LIN {X 0,Y 523.586,Z 1035.497,A -85,B 0,C 180,E1 24820.361,E2 24820.361} C_VEL
LIN {X 0,Y 523.955,Z 1017.547,A -85,B 0,C 180,E1 24819.86,E2 24819.86} C_VEL
LIN {X 0,Y 524.216,Z 988.491,A -85,B 0,C 180,E1 24819.409,E2 24819.409} C_VEL
LIN {X 0,Y 525.099,Z 854.259,A -85,B 0,C 180,E1 24817.476,E2 24817.476} C_VEL
LIN {X 0,Y 524.353,Z 848.699,A -85,B 0,C 180,E1 24817.345,E2 24817.345} C_VEL
LIN {X 0,Y 527.314,Z 813.157,A -85,B 0,C 180,E1 24813.997,E2 24813.997} C_VEL
LIN {X 0,Y 530.511,Z 784.43,A -85,B 0,C 180,E1 24811.152,E2 24811.152} C_VEL
LIN {X 0,Y 534.459,Z 760.277,A -85,B 0,C 180,E1 24808.6,E2 24808.6} C_VEL
LIN {X 0,Y 539.863,Z 738.188,A -85,B 0,C 180,E1 24806.071,E2 24806.071} C_VEL
LIN {X 0,Y 545.29,Z 723.44,A -85,B 0,C 180,E1 24804.202,E2 24804.202} C_VEL
LIN {X 0,Y 548.271,Z 717.496,A -85,B 0,C 180,E1 24803.361,E2 24803.361} C_VEL
LIN {X 0,Y 540.635,Z 729.193,A -85,B 0,C 180,E1 24802.158,E2 24802.158} C_VEL
LIN {X 0,Y 535.477,Z 740.888,A -85,B 0,C 180,E1 24801.051,E2 24801.051} C_VEL
LIN {X 0,Y 532.179,Z 753.467,A -85,B 0,C 180,E1 24799.962,E2 24799.962} C_VEL
LIN {X 0,Y 530.634,Z 767.779,A -85,B 0,C 180,E1 24798.804,E2 24798.804} C_VEL
LIN {X 0,Y 531.093,Z 781.511,A -85,B 0,C 180,E1 24797.721,E2 24797.721} C_VEL
LIN {X 0,Y 533.486,Z 794.423,A -85,B 0,C 180,E1 24796.689,E2 24796.689} C_VEL
LIN {X 0,Y 537.671,Z 806.101,A -85,B 0,C 180,E1 24795.721,E2 24795.721} C_VEL
LIN {X 0,Y 543.177,Z 815.91,A -85,B 0,C 180,E1 24794.872,E2 24794.872} C_VEL
LIN {X 0,Y 550.682,Z 825.132,A -85,B 0,C 180,E1 24794.028,E2 24794.028} C_VEL
LIN {X 0,Y 559.874,Z 833.081,A -85,B 0,C 180,E1 24793.229,E2 24793.229} C_VEL
LIN {X 0,Y 568.972,Z 838.703,A -85,B 0,C 180,E1 24792.582,E2 24792.582} C_VEL
LIN {X 0,Y 573.371,Z 840.473,A -85,B 0,C 180,E1 24792.173,E2 24792.173} C_VEL
LIN {X 0,Y 577.044,Z 841.244,A -85,B 0,C 180,E1 24791.686,E2 24791.686} C_VEL
LIN {X 0,Y 579.923,Z 840.965,A -85,B 0,C 180,E1 24791.111,E2 24791.111} C_VEL
LIN {X 0,Y 581.493,Z 839.74,A -85,B 0,C 180,E1 24790.536,E2 24790.536} C_VEL
LIN {X 0,Y 581.774,Z 837.458,A -85,B 0,C 180,E1 24789.918,E2 24789.918} C_VEL
LIN {X 0,Y 580.503,Z 834.257,A -85,B 0,C 180,E1 24789.335,E2 24789.335} C_VEL
LIN {X 0,Y 577.813,Z 830.456,A -85,B 0,C 180,E1 24788.85,E2 24788.85} C_VEL
LIN {X 0,Y 571.058,Z 821.059,A -85,B 0,C 180,E1 24788,E2 24788} C_VEL
LIN {X 0,Y 565.628,Z 811.116,A -85,B 0,C 180,E1 24787.29,E2 24787.29} C_VEL
LIN {X 0,Y 561.482,Z 850.258,A -85,B 0,C 180,E1 24786.731,E2 24786.731} C_VEL
LIN {X 0,Y 558.358,Z 872.045,A -85,B 0,C 180,E1 24786.299,E2 24786.299} C_VEL
LIN {X 0,Y 556.202,Z 881.325,A -85,B 0,C 180,E1 24785.996,E2 24785.996} C_VEL
LIN {X 0,Y 555.687,Z 885.783,A -85,B 0,C 180,E1 24785.923,E2 24785.923} C_VEL
LIN {X 0,Y 552.428,Z 921.98,A -85,B 0,C 180,E1 24785.512,E2 24785.512} C_VEL
LIN {X 0,Y 548.555,Z 944.063,A -85,B 0,C 180,E1 24785.284,E2 24785.284} C_VEL
LIN {X 0,Y 544.213,Z 961.518,A -85,B 0,C 180,E1 24784.984,E2 24784.984} C_VEL
LIN {X 0,Y 541.11,Z 972.645,A -85,B 0,C 180,E1 24784.625,E2 24784.625} C_VEL
LIN {X 0,Y 540.107,Z 976.205,A -85,B 0,C 180,E1 24784.487,E2 24784.487} C_VEL
LIN {X 0,Y 536.14,Z 989.922,A -85,B 0,C 180,E1 24784.214,E2 24784.214} C_VEL
LIN {X 0,Y 533.243,Z 1000.027,A -85,B 0,C 180,E1 24783.841,E2 24783.841} C_VEL
LIN {X 0,Y 532.563,Z 1003.315,A -85,B 0,C 180,E1 24783.7,E2 24783.7} C_VEL
LIN {X 0,Y 531.76,Z 1066.201,A -85,B 0,C 180,E1 24782.724,E2 24782.724} C_VEL
LIN {X 0,Y 531.071,Z 1087.988,A -85,B 0,C 180,E1 24782.192,E2 24782.192} C_VEL
LIN {X 0,Y 530.194,Z 1110.298,A -85,B 0,C 180,E1 24781.429,E2 24781.429} C_VEL
LIN {X 0,Y 529.157,Z 1131.269,A -85,B 0,C 180,E1 24780.501,E2 24780.501} C_VEL
LIN {X 0,Y 528.011,Z 1151.791,A -85,B 0,C 180,E1 24779.371,E2 24779.371} C_VEL
LIN {X 0,Y 526.773,Z 1171.709,A -85,B 0,C 180,E1 24778.042,E2 24778.042} C_VEL
LIN {X 0,Y 525.528,Z 1191.133,A -85,B 0,C 180,E1 24776.498,E2 24776.498} C_VEL
LIN {X 0,Y 524.371,Z 1208.653,A -85,B 0,C 180,E1 24774.857,E2 24774.857} C_VEL
LIN {X 0,Y 523.398,Z 1223.625,A -85,B 0,C 180,E1 24773.24,E2 24773.24} C_VEL
LIN {X 0,Y 522.415,Z 1239.904,A -85,B 0,C 180,E1 24771.207,E2 24771.207} C_VEL
LIN {X 0,Y 521.625,Z 1254.014,A -85,B 0,C 180,E1 24769.134,E2 24769.134} C_VEL
LIN {X 0,Y 521.016,Z 1266.743,A -85,B 0,C 180,E1 24766.96,E2 24766.96} C_VEL
LIN {X 0,Y 520.548,Z 1277.844,A -85,B 0,C 180,E1 24764.688,E2 24764.688} C_VEL
LIN {X 0,Y 520.249,Z 1287.1,A -85,B 0,C 180,E1 24762.431,E2 24762.431} C_VEL
LIN {X 0,Y 520.058,Z 1295.215,A -85,B 0,C 180,E1 24759.965,E2 24759.965} C_VEL
LIN {X 0,Y 519.971,Z 1300.895,A -85,B 0,C 180,E1 24757.736,E2 24757.736} C_VEL
LIN {X 0,Y 519.921,Z 1305.493,A -85,B 0,C 180,E1 24755.297,E2 24755.297} C_VEL
LIN {X 0,Y 519.902,Z 1308.295,A -85,B 0,C 180,E1 24752.867,E2 24752.867} C_VEL
LIN {X 0,Y 519.896,Z 1309.373,A -85,B 0,C 180,E1 24750.662,E2 24750.662} C_VEL
LIN {X 0,Y 519.896,Z 1309.038,A -85,B 0,C 180,E1 24748.237,E2 24748.237} C_VEL
LIN {X 0,Y 519.905,Z 1307.108,A -85,B 0,C 180,E1 24745.92,E2 24745.92} C_VEL
LIN {X 0,Y 519.931,Z 1303.619,A -85,B 0,C 180,E1 24743.597,E2 24743.597} C_VEL
LIN {X 0,Y 519.999,Z 1298.291,A -85,B 0,C 180,E1 24741.152,E2 24741.152} C_VEL
LIN {X 0,Y 520.135,Z 1291.394,A -85,B 0,C 180,E1 24738.805,E2 24738.805} C_VEL
LIN {X 0,Y 520.382,Z 1282.793,A -85,B 0,C 180,E1 24736.463,E2 24736.463} C_VEL
LIN {X 0,Y 520.771,Z 1271.951,A -85,B 0,C 180,E1 24734.065,E2 24734.065} C_VEL
LIN {X 0,Y 521.239,Z 1261.598,A -85,B 0,C 180,E1 24732.127,E2 24732.127} C_VEL
LIN {X 0,Y 521.949,Z 1248.058,A -85,B 0,C 180,E1 24729.947,E2 24729.947} C_VEL
LIN {X 0,Y 522.774,Z 1233.701,A -85,B 0,C 180,E1 24727.984,E2 24727.984} C_VEL
LIN {X 0,Y 523.673,Z 1219.46,A -85,B 0,C 180,E1 24726.288,E2 24726.288} C_VEL
LIN {X 0,Y 524.839,Z 1201.727,A -85,B 0,C 180,E1 24724.459,E2 24724.459} C_VEL
LIN {X 0,Y 526.047,Z 1182.855,A -85,B 0,C 180,E1 24722.814,E2 24722.814} C_VEL
LIN {X 0,Y 527.349,Z 1162.825,A -85,B 0,C 180,E1 24721.336,E2 24721.336} C_VEL
LIN {X 0,Y 528.528,Z 1142.749,A -85,B 0,C 180,E1 24720.101,E2 24720.101} C_VEL
LIN {X 0,Y 529.657,Z 1121.584,A -85,B 0,C 180,E1 24719.043,E2 24719.043} C_VEL
LIN {X 0,Y 530.645,Z 1099.656,A -85,B 0,C 180,E1 24718.181,E2 24718.181} C_VEL
LIN {X 0,Y 531.428,Z 1077.651,A -85,B 0,C 180,E1 24717.53,E2 24717.53} C_VEL
LIN {X 0,Y 531.973,Z 1055.21,A -85,B 0,C 180,E1 24717.082,E2 24717.082} C_VEL
LIN {X 0,Y 532.624,Z 1002.328,A -85,B 0,C 180,E1 24716.277,E2 24716.277} C_VEL
LIN {X 0,Y 535.397,Z 992.455,A -85,B 0,C 180,E1 24715.863,E2 24715.863} C_VEL
LIN {X 0,Y 539.286,Z 979.138,A -85,B 0,C 180,E1 24715.554,E2 24715.554} C_VEL
LIN {X 0,Y 540.609,Z 974.405,A -85,B 0,C 180,E1 24715.46,E2 24715.46} C_VEL
LIN {X 0,Y 543.293,Z 964.872,A -85,B 0,C 180,E1 24715.102,E2 24715.102} C_VEL
LIN {X 0,Y 547.461,Z 948.839,A -85,B 0,C 180,E1 24714.78,E2 24714.78} C_VEL
LIN {X 0,Y 551.573,Z 927.951,A -85,B 0,C 180,E1 24714.547,E2 24714.547} C_VEL
LIN {X 0,Y 554.193,Z 904.712,A -85,B 0,C 180,E1 24714.291,E2 24714.291} C_VEL
LIN {X 0,Y 556.16,Z 881.458,A -85,B 0,C 180,E1 24714.01,E2 24714.01} C_VEL
LIN {X 0,Y 558.316,Z 872.279,A -85,B 0,C 180,E1 24713.707,E2 24713.707} C_VEL
LIN {X 0,Y 561.42,Z 850.756,A -85,B 0,C 180,E1 24713.277,E2 24713.277} C_VEL
LIN {X 0,Y 565.558,Z 811.884,A -85,B 0,C 180,E1 24712.719,E2 24712.719} C_VEL
LIN {X 0,Y 565.709,Z 810.985,A -85,B 0,C 180,E1 24712.699,E2 24712.699} C_VEL
LIN {X 0,Y 571.284,Z 821.421,A -85,B 0,C 180,E1 24711.971,E2 24711.971} C_VEL
LIN {X 0,Y 577.959,Z 830.632,A -85,B 0,C 180,E1 24711.131,E2 24711.131} C_VEL
LIN {X 0,Y 580.567,Z 834.367,A -85,B 0,C 180,E1 24710.648,E2 24710.648} C_VEL
LIN {X 0,Y 581.789,Z 837.556,A -85,B 0,C 180,E1 24710.061,E2 24710.061} C_VEL
LIN {X 0,Y 581.489,Z 839.748,A -85,B 0,C 180,E1 24709.462,E2 24709.462} C_VEL
LIN {X 0,Y 579.921,Z 840.971,A -85,B 0,C 180,E1 24708.889,E2 24708.889} C_VEL
LIN {X 0,Y 577.042,Z 841.249,A -85,B 0,C 180,E1 24708.314,E2 24708.314} C_VEL
LIN {X 0,Y 573.37,Z 840.478,A -85,B 0,C 180,E1 24707.827,E2 24707.827} C_VEL
LIN {X 0,Y 564.453,Z 836.474,A -85,B 0,C 180,E1 24706.87,E2 24706.87} C_VEL
LIN {X 0,Y 556.319,Z 830.523,A -85,B 0,C 180,E1 24705.816,E2 24705.816} C_VEL
LIN {X 0,Y 549.697,Z 823.015,A -85,B 0,C 180,E1 24704.742,E2 24704.742} C_VEL
LIN {X 0,Y 544.58,Z 813.966,A -85,B 0,C 180,E1 24703.657,E2 24703.657} C_VEL
LIN {X 0,Y 540.972,Z 803.368,A -85,B 0,C 180,E1 24702.568,E2 24702.568} C_VEL
LIN {X 0,Y 538.865,Z 790.955,A -85,B 0,C 180,E1 24701.444,E2 24701.444} C_VEL
LIN {X 0,Y 538.28,Z 775.777,A -85,B 0,C 180,E1 24700.233,E2 24700.233} C_VEL
LIN {X 0,Y 541.066,Z 725.504,A -85,B 0,C 180,E1 24696.581,E2 24696.581} C_VEL
LIN {X 0,Y 541.898,Z 709.421,A -85,B 0,C 180,E1 24695.361,E2 24695.361} C_VEL
LIN {X 0,Y 533.055,Z 693.053,A -85,B 0,C 180,E1 24692.825,E2 24692.825} C_VEL
LIN {X 0,Y 527.803,Z 683.663,A -85,B 0,C 180,E1 24691.269,E2 24691.269} C_VEL
LIN {X 0,Y 525.459,Z 679.281,A -85,B 0,C 180,E1 24690.534,E2 24690.534} C_VEL
LIN {X 0,Y 523.439,Z 675.653,A -85,B 0,C 180,E1 24689.904,E2 24689.904} C_VEL
LIN {X 0,Y 522.358,Z 673.996,A -85,B 0,C 180,E1 24689.593,E2 24689.593} C_VEL
LIN {X 0,Y 520.765,Z 670.882,A -85,B 0,C 180,E1 24689.062,E2 24689.062} C_VEL
LIN {X 0,Y 520.584,Z 669.89,A -85,B 0,C 180,E1 24688.904,E2 24688.904} C_VEL
LIN {X 0,Y 520.583,Z 669.888,A -85,B 0,C 180,E1 24685.36,E2 24685.36} C_VEL
LIN {X 0,Y 520.582,Z 669.887,A -85,B 0,C 180,E1 24681.876,E2 24681.876} C_VEL
LIN {X 0,Y 520.574,Z 669.89,A -85,B 0,C 180,E1 24678.413,E2 24678.413} C_VEL
LIN {X 0,Y 520.583,Z 669.892,A -85,B 0,C 180,E1 24674.967,E2 24674.967} C_VEL
LIN {X 0,Y 520.588,Z 669.889,A -85,B 0,C 180,E1 24671.41,E2 24671.41} C_VEL
LIN {X 0,Y 520.576,Z 669.889,A -85,B 0,C 180,E1 24667.837,E2 24667.837} C_VEL
LIN {X 0,Y 520.586,Z 669.889,A -85,B 0,C 180,E1 24664.406,E2 24664.406} C_VEL
LIN {X 0,Y 520.586,Z 669.888,A -85,B 0,C 180,E1 24660.88,E2 24660.88} C_VEL
LIN {X 0,Y 520.582,Z 669.889,A -85,B 0,C 180,E1 24657.358,E2 24657.358} C_VEL
LIN {X 0,Y 520.587,Z 669.889,A -85,B 0,C 180,E1 24653.825,E2 24653.825} C_VEL
LIN {X 0,Y 520.587,Z 669.892,A -85,B 0,C 180,E1 24650.269,E2 24650.269} C_VEL
LIN {X 0,Y 520.577,Z 669.888,A -85,B 0,C 180,E1 24646.787,E2 24646.787} C_VEL
LIN {X 0,Y 520.587,Z 669.888,A -85,B 0,C 180,E1 24643.256,E2 24643.256} C_VEL
LIN {X 0,Y 520.582,Z 669.888,A -85,B 0,C 180,E1 24639.657,E2 24639.657} C_VEL
LIN {X 0,Y 520.574,Z 669.889,A -85,B 0,C 180,E1 24636.212,E2 24636.212} C_VEL
LIN {X 0,Y 520.581,Z 669.879,A -85,B 0,C 180,E1 24632.779,E2 24632.779} C_VEL
LIN {X 0,Y 520.589,Z 669.881,A -85,B 0,C 180,E1 24629.277,E2 24629.277} C_VEL
LIN {X 0,Y 520.588,Z 669.876,A -85,B 0,C 180,E1 24625.754,E2 24625.754} C_VEL
LIN {X 0,Y 520.581,Z 669.892,A -85,B 0,C 180,E1 24622.307,E2 24622.307} C_VEL
LIN {X 0,Y 520.571,Z 669.873,A -85,B 0,C 180,E1 24618.842,E2 24618.842} C_VEL
LIN {X 0,Y 520.585,Z 669.882,A -85,B 0,C 180,E1 24617.879,E2 24617.879} C_VEL
LIN {X 0,Y 519.613,Z 670.014,A -85,B 0,C 180,E1 24617.032,E2 24617.032} C_VEL
LIN {X 0,Y 513.091,Z 670.826,A -85,B 0,C 180,E1 24614.588,E2 24614.588} C_VEL
LIN {X 0,Y 512.64,Z 670.882,A -85,B 0,C 180,E1 24614.028,E2 24614.028} C_VEL
LIN {X 0,Y 512.679,Z 671.112,A -85,B 0,C 180,E1 24610.616,E2 24610.616} C_VEL
LIN {X 0,Y 513.821,Z 674.165,A -85,B 0,C 180,E1 24610.288,E2 24610.288} C_VEL
LIN {X 0,Y 522.026,Z 692.981,A -85,B 0,C 180,E1 24608.163,E2 24608.163} C_VEL
LIN {X 0,Y 524.698,Z 700.431,A -85,B 0,C 180,E1 24607.379,E2 24607.379} C_VEL
LIN {X 0,Y 522.968,Z 748.227,A -85,B 0,C 180,E1 24604.002,E2 24604.002} C_VEL
LIN {X 0,Y 522.481,Z 768.097,A -85,B 0,C 180,E1 24602.665,E2 24602.665} C_VEL
LIN {X 0,Y 524.515,Z 781.949,A -85,B 0,C 180,E1 24602.299,E2 24602.299} C_VEL
LIN {X 0,Y 521.936,Z 1016.462,A -85,B 0,C 180,E1 24598.79,E2 24598.79} C_VEL
LIN {X 0,Y 521.472,Z 1038.136,A -85,B 0,C 180,E1 24598.367,E2 24598.367} C_VEL
LIN {X 0,Y 520.771,Z 1058.877,A -85,B 0,C 180,E1 24597.752,E2 24597.752} C_VEL
LIN {X 0,Y 519.953,Z 1077.833,A -85,B 0,C 180,E1 24596.988,E2 24596.988} C_VEL
LIN {X 0,Y 519.007,Z 1096.138,A -85,B 0,C 180,E1 24596.055,E2 24596.055} C_VEL
LIN {X 0,Y 517.914,Z 1115.556,A -85,B 0,C 180,E1 24594.833,E2 24594.833} C_VEL
LIN {X 0,Y 516.831,Z 1133.209,A -85,B 0,C 180,E1 24593.485,E2 24593.485} C_VEL
LIN {X 0,Y 515.776,Z 1149.876,A -85,B 0,C 180,E1 24591.971,E2 24591.971} C_VEL
LIN {X 0,Y 514.806,Z 1165.721,A -85,B 0,C 180,E1 24590.267,E2 24590.267} C_VEL
LIN {X 0,Y 513.937,Z 1180.619,A -85,B 0,C 180,E1 24588.37,E2 24588.37} C_VEL
LIN {X 0,Y 513.248,Z 1193.625,A -85,B 0,C 180,E1 24586.407,E2 24586.407} C_VEL
LIN {X 0,Y 512.723,Z 1205.136,A -85,B 0,C 180,E1 24584.339,E2 24584.339} C_VEL
LIN {X 0,Y 512.365,Z 1214.674,A -85,B 0,C 180,E1 24582.281,E2 24582.281} C_VEL
LIN {X 0,Y 512.118,Z 1223.218,A -85,B 0,C 180,E1 24580.006,E2 24580.006} C_VEL
LIN {X 0,Y 511.993,Z 1229.79,A -85,B 0,C 180,E1 24577.744,E2 24577.744} C_VEL
LIN {X 0,Y 511.93,Z 1234.587,A -85,B 0,C 180,E1 24575.491,E2 24575.491} C_VEL
LIN {X 0,Y 511.913,Z 1237.847,A -85,B 0,C 180,E1 24573.135,E2 24573.135} C_VEL
LIN {X 0,Y 511.91,Z 1239.341,A -85,B 0,C 180,E1 24570.783,E2 24570.783} C_VEL
LIN {X 0,Y 511.9,Z 1239.167,A -85,B 0,C 180,E1 24568.545,E2 24568.545} C_VEL
LIN {X 0,Y 511.911,Z 1237.374,A -85,B 0,C 180,E1 24566.304,E2 24566.304} C_VEL
LIN {X 0,Y 511.938,Z 1233.93,A -85,B 0,C 180,E1 24564.058,E2 24564.058} C_VEL
LIN {X 0,Y 511.996,Z 1228.822,A -85,B 0,C 180,E1 24561.804,E2 24561.804} C_VEL
LIN {X 0,Y 512.143,Z 1221.931,A -85,B 0,C 180,E1 24559.539,E2 24559.539} C_VEL
LIN {X 0,Y 512.406,Z 1213.59,A -85,B 0,C 180,E1 24557.376,E2 24557.376} C_VEL
LIN {X 0,Y 512.812,Z 1203.268,A -85,B 0,C 180,E1 24555.201,E2 24555.201} C_VEL
LIN {X 0,Y 513.373,Z 1191.365,A -85,B 0,C 180,E1 24553.13,E2 24553.13} C_VEL
LIN {X 0,Y 514.102,Z 1177.909,A -85,B 0,C 180,E1 24551.164,E2 24551.164} C_VEL
LIN {X 0,Y 514.959,Z 1163.358,A -85,B 0,C 180,E1 24549.369,E2 24549.369} C_VEL
LIN {X 0,Y 515.916,Z 1147.72,A -85,B 0,C 180,E1 24547.73,E2 24547.73} C_VEL
LIN {X 0,Y 516.976,Z 1130.589,A -85,B 0,C 180,E1 24546.212,E2 24546.212} C_VEL
LIN {X 0,Y 518.063,Z 1112.527,A -85,B 0,C 180,E1 24544.874,E2 24544.874} C_VEL
LIN {X 0,Y 519.112,Z 1094.057,A -85,B 0,C 180,E1 24543.742,E2 24543.742} C_VEL
LIN {X 0,Y 520.077,Z 1075.446,A -85,B 0,C 180,E1 24542.809,E2 24542.809} C_VEL
LIN {X 0,Y 520.934,Z 1055.241,A -85,B 0,C 180,E1 24542.031,E2 24542.031} C_VEL
LIN {X 0,Y 521.55,Z 1035.024,A -85,B 0,C 180,E1 24541.467,E2 24541.467} C_VEL
LIN {X 0,Y 521.988,Z 1011.53,A -85,B 0,C 180,E1 24541.047,E2 24541.047} C_VEL
LIN {X 0,Y 524.463,Z 786.209,A -85,B 0,C 180,E1 24537.676,E2 24537.676} C_VEL
LIN {X 0,Y 520.542,Z 769.078,A -85,B 0,C 180,E1 24537.101,E2 24537.101} C_VEL
LIN {X 0,Y 521.787,Z 734.75,A -85,B 0,C 180,E1 24533.693,E2 24533.693} C_VEL
LIN {X 0,Y 523.14,Z 702.195,A -85,B 0,C 180,E1 24530.33,E2 24530.33} C_VEL
LIN {X 0,Y 523.014,Z 698.905,A -85,B 0,C 180,E1 24529.965,E2 24529.965} C_VEL
LIN {X 0,Y 517.23,Z 683.066,A -85,B 0,C 180,E1 24527.764,E2 24527.764} C_VEL
LIN {X 0,Y 512.646,Z 670.881,A -85,B 0,C 180,E1 24526.029,E2 24526.029} C_VEL
LIN {X 0,Y 512.648,Z 670.874,A -85,B 0,C 180,E1 24522.441,E2 24522.441} C_VEL
LIN {X 0,Y 512.633,Z 670.88,A -85,B 0,C 180,E1 24518.901,E2 24518.901} C_VEL
LIN {X 0,Y 512.659,Z 671.045,A -85,B 0,C 180,E1 24517.711,E2 24517.711} C_VEL
LIN {X 0,Y 521.567,Z 693.534,A -85,B 0,C 180,E1 24514.673,E2 24514.673} C_VEL
LIN {X 0,Y 523.379,Z 698.995,A -85,B 0,C 180,E1 24513.992,E2 24513.992} C_VEL
LIN {X 0,Y 521.452,Z 736.924,A -85,B 0,C 180,E1 24510.578,E2 24510.578} C_VEL
LIN {X 0,Y 519.575,Z 775.825,A -85,B 0,C 180,E1 24507.135,E2 24507.135} C_VEL
LIN {X 0,Y 517.753,Z 816.666,A -85,B 0,C 180,E1 24503.563,E2 24503.563} C_VEL
LIN {X 0,Y 516.554,Z 847.209,A -85,B 0,C 180,E1 24500.942,E2 24500.942} C_VEL
LIN {X 0,Y 517.783,Z 857.852,A -85,B 0,C 180,E1 24500.712,E2 24500.712} C_VEL
LIN {X 0,Y 516.46,Z 1013.64,A -85,B 0,C 180,E1 24498.42,E2 24498.42} C_VEL
LIN {X 0,Y 516.179,Z 1028.414,A -85,B 0,C 180,E1 24498.07,E2 24498.07} C_VEL
LIN {X 0,Y 515.773,Z 1045.052,A -85,B 0,C 180,E1 24497.487,E2 24497.487} C_VEL
LIN {X 0,Y 515.244,Z 1060.015,A -85,B 0,C 180,E1 24496.755,E2 24496.755} C_VEL
LIN {X 0,Y 514.717,Z 1073.391,A -85,B 0,C 180,E1 24495.938,E2 24495.938} C_VEL
LIN {X 0,Y 514.224,Z 1085.53,A -85,B 0,C 180,E1 24495.045,E2 24495.045} C_VEL
LIN {X 0,Y 513.688,Z 1099.05,A -85,B 0,C 180,E1 24493.852,E2 24493.852} C_VEL
LIN {X 0,Y 513.16,Z 1111.489,A -85,B 0,C 180,E1 24492.491,E2 24492.491} C_VEL
LIN {X 0,Y 512.787,Z 1121.038,A -85,B 0,C 180,E1 24491.244,E2 24491.244} C_VEL
LIN {X 0,Y 512.477,Z 1129.824,A -85,B 0,C 180,E1 24489.886,E2 24489.886} C_VEL
LIN {X 0,Y 512.244,Z 1137.749,A -85,B 0,C 180,E1 24488.418,E2 24488.418} C_VEL
LIN {X 0,Y 512.053,Z 1145.975,A -85,B 0,C 180,E1 24486.503,E2 24486.503} C_VEL
LIN {X 0,Y 511.965,Z 1151.39,A -85,B 0,C 180,E1 24484.818,E2 24484.818} C_VEL
LIN {X 0,Y 511.928,Z 1155.154,A -85,B 0,C 180,E1 24483.247,E2 24483.247} C_VEL
LIN {X 0,Y 511.917,Z 1157.862,A -85,B 0,C 180,E1 24481.567,E2 24481.567} C_VEL
LIN {X 0,Y 511.917,Z 1159.404,A -85,B 0,C 180,E1 24479.553,E2 24479.553} C_VEL
LIN {X 0,Y 511.914,Z 1159.026,A -85,B 0,C 180,E1 24477.65,E2 24477.65} C_VEL
LIN {X 0,Y 511.916,Z 1157.362,A -85,B 0,C 180,E1 24475.968,E2 24475.968} C_VEL
LIN {X 0,Y 511.936,Z 1154.161,A -85,B 0,C 180,E1 24474.171,E2 24474.171} C_VEL
LIN {X 0,Y 512.006,Z 1148.521,A -85,B 0,C 180,E1 24472.143,E2 24472.143} C_VEL
LIN {X 0,Y 512.124,Z 1142.576,A -85,B 0,C 180,E1 24470.561,E2 24470.561} C_VEL
LIN {X 0,Y 512.301,Z 1135.702,A -85,B 0,C 180,E1 24469.087,E2 24469.087} C_VEL
LIN {X 0,Y 512.595,Z 1126.677,A -85,B 0,C 180,E1 24467.496,E2 24467.496} C_VEL
LIN {X 0,Y 513.002,Z 1115.365,A -85,B 0,C 180,E1 24465.899,E2 24465.899} C_VEL
LIN {X 0,Y 513.434,Z 1104.609,A -85,B 0,C 180,E1 24464.642,E2 24464.642} C_VEL
LIN {X 0,Y 513.89,Z 1093.87,A -85,B 0,C 180,E1 24463.58,E2 24463.58} C_VEL
LIN {X 0,Y 514.421,Z 1081.215,A -85,B 0,C 180,E1 24462.525,E2 24462.525} C_VEL
LIN {X 0,Y 515.068,Z 1065.082,A -85,B 0,C 180,E1 24461.437,E2 24461.437} C_VEL
LIN {X 0,Y 515.536,Z 1052.287,A -85,B 0,C 180,E1 24460.749,E2 24460.749} C_VEL
LIN {X 0,Y 515.956,Z 1038.76,A -85,B 0,C 180,E1 24460.177,E2 24460.177} C_VEL
LIN {X 0,Y 516.304,Z 1024.146,A -85,B 0,C 180,E1 24459.718,E2 24459.718} C_VEL
LIN {X 0,Y 516.581,Z 1005.675,A -85,B 0,C 180,E1 24459.35,E2 24459.35} C_VEL
LIN {X 0,Y 517.754,Z 885.861,A -85,B 0,C 180,E1 24457.559,E2 24457.559} C_VEL
LIN {X 0,Y 517.956,Z 854.586,A -85,B 0,C 180,E1 24457.053,E2 24457.053} C_VEL
LIN {X 0,Y 517.652,Z 851.854,A -85,B 0,C 180,E1 24456.975,E2 24456.975} C_VEL
LIN {X 0,Y 518.629,Z 841.769,A -85,B 0,C 180,E1 24456.039,E2 24456.039} C_VEL
LIN {X 0,Y 521.516,Z 811.449,A -85,B 0,C 180,E1 24453.098,E2 24453.098} C_VEL
LIN {X 0,Y 525.436,Z 782.786,A -85,B 0,C 180,E1 24450.165,E2 24450.165} C_VEL
LIN {X 0,Y 530.708,Z 757.235,A -85,B 0,C 180,E1 24447.333,E2 24447.333} C_VEL
LIN {X 0,Y 536.128,Z 739.728,A -85,B 0,C 180,E1 24445.203,E2 24445.203} C_VEL
LIN {X 0,Y 541.891,Z 727.063,A -85,B 0,C 180,E1 24443.511,E2 24443.511} C_VEL
LIN {X 0,Y 541.923,Z 726.971,A -85,B 0,C 180,E1 24443.475,E2 24443.475} C_VEL
LIN {X 0,Y 534.369,Z 738.425,A -85,B 0,C 180,E1 24442.277,E2 24442.277} C_VEL
LIN {X 0,Y 529.068,Z 750.147,A -85,B 0,C 180,E1 24441.135,E2 24441.135} C_VEL
LIN {X 0,Y 525.792,Z 762.558,A -85,B 0,C 180,E1 24440.003,E2 24440.003} C_VEL
LIN {X 0,Y 524.433,Z 775.763,A -85,B 0,C 180,E1 24438.859,E2 24438.859} C_VEL
LIN {X 0,Y 525.068,Z 788.685,A -85,B 0,C 180,E1 24437.763,E2 24437.763} C_VEL
LIN {X 0,Y 527.72,Z 801.303,A -85,B 0,C 180,E1 24436.682,E2 24436.682} C_VEL
LIN {X 0,Y 532.247,Z 812.841,A -85,B 0,C 180,E1 24435.668,E2 24435.668} C_VEL
LIN {X 0,Y 538.091,Z 822.524,A -85,B 0,C 180,E1 24434.78,E2 24434.78} C_VEL
LIN {X 0,Y 545.622,Z 831.387,A -85,B 0,C 180,E1 24433.931,E2 24433.931} C_VEL
LIN {X 0,Y 554.841,Z 839.222,A -85,B 0,C 180,E1 24433.128,E2 24433.128} C_VEL
LIN {X 0,Y 565.649,Z 845.773,A -85,B 0,C 180,E1 24432.365,E2 24432.365} C_VEL
LIN {X 0,Y 570.231,Z 847.6,A -85,B 0,C 180,E1 24431.974,E2 24431.974} C_VEL
LIN {X 0,Y 574.077,Z 848.447,A -85,B 0,C 180,E1 24431.503,E2 24431.503} C_VEL
LIN {X 0,Y 577.149,Z 848.29,A -85,B 0,C 180,E1 24430.946,E2 24430.946} C_VEL
LIN {X 0,Y 579.007,Z 847.156,A -85,B 0,C 180,E1 24430.359,E2 24430.359} C_VEL
LIN {X 0,Y 579.537,Z 845.005,A -85,B 0,C 180,E1 24429.733,E2 24429.733} C_VEL
LIN {X 0,Y 578.525,Z 841.971,A -85,B 0,C 180,E1 24429.143,E2 24429.143} C_VEL
LIN {X 0,Y 576.062,Z 838.338,A -85,B 0,C 180,E1 24428.639,E2 24428.639} C_VEL
LIN {X 0,Y 569.216,Z 829.275,A -85,B 0,C 180,E1 24427.762,E2 24427.762} C_VEL
LIN {X 0,Y 568.815,Z 828.887,A -85,B 0,C 180,E1 24427.71,E2 24427.71} C_VEL
LIN {X 0,Y 564.788,Z 862.62,A -85,B 0,C 180,E1 24427.178,E2 24427.178} C_VEL
LIN {X 0,Y 562.023,Z 878.875,A -85,B 0,C 180,E1 24426.805,E2 24426.805} C_VEL
LIN {X 0,Y 560.473,Z 885.57,A -85,B 0,C 180,E1 24426.593,E2 24426.593} C_VEL
LIN {X 0,Y 557.992,Z 907.178,A -85,B 0,C 180,E1 24426.403,E2 24426.403} C_VEL
LIN {X 0,Y 553.45,Z 929.367,A -85,B 0,C 180,E1 24426.247,E2 24426.247} C_VEL
LIN {X 0,Y 547.519,Z 949.909,A -85,B 0,C 180,E1 24426.05,E2 24426.05} C_VEL
LIN {X 0,Y 542.494,Z 965.172,A -85,B 0,C 180,E1 24425.751,E2 24425.751} C_VEL
LIN {X 0,Y 539.344,Z 975.29,A -85,B 0,C 180,E1 24425.403,E2 24425.403} C_VEL
LIN {X 0,Y 538.465,Z 978.104,A -85,B 0,C 180,E1 24425.307,E2 24425.307} C_VEL
LIN {X 0,Y 533.481,Z 991.991,A -85,B 0,C 180,E1 24424.996,E2 24424.996} C_VEL
LIN {X 0,Y 530.187,Z 1002.66,A -85,B 0,C 180,E1 24424.586,E2 24424.586} C_VEL
LIN {X 0,Y 526.007,Z 1016.588,A -85,B 0,C 180,E1 24424.022,E2 24424.022} C_VEL
LIN {X 0,Y 525.716,Z 1019.219,A -85,B 0,C 180,E1 24423.943,E2 24423.943} C_VEL
LIN {X 0,Y 525.011,Z 1066.716,A -85,B 0,C 180,E1 24423.186,E2 24423.186} C_VEL
LIN {X 0,Y 524.259,Z 1088.479,A -85,B 0,C 180,E1 24422.646,E2 24422.646} C_VEL
LIN {X 0,Y 523.315,Z 1110.292,A -85,B 0,C 180,E1 24421.89,E2 24421.89} C_VEL
LIN {X 0,Y 522.179,Z 1131.351,A -85,B 0,C 180,E1 24420.948,E2 24420.948} C_VEL
LIN {X 0,Y 520.917,Z 1151.797,A -85,B 0,C 180,E1 24419.811,E2 24419.811} C_VEL
LIN {X 0,Y 519.54,Z 1171.996,A -85,B 0,C 180,E1 24418.445,E2 24418.445} C_VEL
LIN {X 0,Y 518.136,Z 1191.806,A -85,B 0,C 180,E1 24416.844,E2 24416.844} C_VEL
LIN {X 0,Y 516.901,Z 1208.564,A -85,B 0,C 180,E1 24415.25,E2 24415.25} C_VEL
LIN {X 0,Y 515.828,Z 1223.672,A -85,B 0,C 180,E1 24413.595,E2 24413.595} C_VEL
LIN {X 0,Y 514.708,Z 1240.27,A -85,B 0,C 180,E1 24411.489,E2 24411.489} C_VEL
LIN {X 0,Y 513.845,Z 1254.008,A -85,B 0,C 180,E1 24409.435,E2 24409.435} C_VEL
LIN {X 0,Y 513.155,Z 1266.743,A -85,B 0,C 180,E1 24407.228,E2 24407.228} C_VEL
LIN {X 0,Y 512.625,Z 1277.839,A -85,B 0,C 180,E1 24404.92,E2 24404.92} C_VEL
LIN {X 0,Y 512.289,Z 1287.154,A -85,B 0,C 180,E1 24402.613,E2 24402.613} C_VEL
LIN {X 0,Y 512.079,Z 1295.212,A -85,B 0,C 180,E1 24400.122,E2 24400.122} C_VEL
LIN {X 0,Y 511.977,Z 1300.643,A -85,B 0,C 180,E1 24397.971,E2 24397.971} C_VEL
LIN {X 0,Y 511.93,Z 1305.167,A -85,B 0,C 180,E1 24395.605,E2 24395.605} C_VEL
LIN {X 0,Y 511.906,Z 1308.209,A -85,B 0,C 180,E1 24393.023,E2 24393.023} C_VEL
LIN {X 0,Y 511.899,Z 1309.347,A -85,B 0,C 180,E1 24390.784,E2 24390.784} C_VEL
LIN {X 0,Y 511.895,Z 1309.154,A -85,B 0,C 180,E1 24388.434,E2 24388.434} C_VEL
LIN {X 0,Y 511.903,Z 1307.242,A -85,B 0,C 180,E1 24385.968,E2 24385.968} C_VEL
LIN {X 0,Y 511.932,Z 1303.812,A -85,B 0,C 180,E1 24383.609,E2 24383.609} C_VEL
LIN {X 0,Y 512.007,Z 1298.681,A -85,B 0,C 180,E1 24381.161,E2 24381.161} C_VEL
LIN {X 0,Y 512.156,Z 1291.762,A -85,B 0,C 180,E1 24378.743,E2 24378.743} C_VEL
LIN {X 0,Y 512.43,Z 1283.145,A -85,B 0,C 180,E1 24376.336,E2 24376.336} C_VEL
LIN {X 0,Y 512.858,Z 1272.524,A -85,B 0,C 180,E1 24373.929,E2 24373.929} C_VEL
LIN {X 0,Y 513.403,Z 1261.763,A -85,B 0,C 180,E1 24371.875,E2 24371.875} C_VEL
LIN {X 0,Y 514.16,Z 1248.839,A -85,B 0,C 180,E1 24369.749,E2 24369.749} C_VEL
LIN {X 0,Y 515.07,Z 1234.614,A -85,B 0,C 180,E1 24367.758,E2 24367.758} C_VEL
LIN {X 0,Y 516.041,Z 1220.611,A -85,B 0,C 180,E1 24366.052,E2 24366.052} C_VEL
LIN {X 0,Y 517.302,Z 1203.349,A -85,B 0,C 180,E1 24364.223,E2 24364.223} C_VEL
LIN {X 0,Y 518.617,Z 1184.872,A -85,B 0,C 180,E1 24362.564,E2 24362.564} C_VEL
LIN {X 0,Y 520.012,Z 1165.375,A -85,B 0,C 180,E1 24361.082,E2 24361.082} C_VEL
LIN {X 0,Y 521.274,Z 1145.785,A -85,B 0,C 180,E1 24359.832,E2 24359.832} C_VEL
LIN {X 0,Y 522.529,Z 1125.443,A -85,B 0,C 180,E1 24358.765,E2 24358.765} C_VEL
LIN {X 0,Y 523.628,Z 1103.794,A -85,B 0,C 180,E1 24357.858,E2 24357.858} C_VEL
LIN {X 0,Y 524.537,Z 1081.939,A -85,B 0,C 180,E1 24357.17,E2 24357.17} C_VEL
LIN {X 0,Y 525.152,Z 1060.11,A -85,B 0,C 180,E1 24356.689,E2 24356.689} C_VEL
LIN {X 0,Y 525.837,Z 1017.266,A -85,B 0,C 180,E1 24356.012,E2 24356.012} C_VEL
LIN {X 0,Y 528.869,Z 1006.939,A -85,B 0,C 180,E1 24355.579,E2 24355.579} C_VEL
LIN {X 0,Y 530.73,Z 1000.702,A -85,B 0,C 180,E1 24355.324,E2 24355.324} C_VEL
LIN {X 0,Y 534.294,Z 989.632,A -85,B 0,C 180,E1 24354.936,E2 24354.936} C_VEL
LIN {X 0,Y 539.067,Z 976.277,A -85,B 0,C 180,E1 24354.642,E2 24354.642} C_VEL
LIN {X 0,Y 542.08,Z 966.441,A -85,B 0,C 180,E1 24354.284,E2 24354.284} C_VEL
LIN {X 0,Y 547.241,Z 950.774,A -85,B 0,C 180,E1 24353.963,E2 24353.963} C_VEL
LIN {X 0,Y 553.168,Z 930.485,A -85,B 0,C 180,E1 24353.761,E2 24353.761} C_VEL
LIN {X 0,Y 557.819,Z 908.253,A -85,B 0,C 180,E1 24353.605,E2 24353.605} C_VEL
LIN {X 0,Y 560.385,Z 886.737,A -85,B 0,C 180,E1 24353.42,E2 24353.42} C_VEL
LIN {X 0,Y 560.86,Z 883.521,A -85,B 0,C 180,E1 24353.354,E2 24353.354} C_VEL
LIN {X 0,Y 563.275,Z 872.39,A -85,B 0,C 180,E1 24353.025,E2 24353.025} C_VEL
LIN {X 0,Y 566.675,Z 848.028,A -85,B 0,C 180,E1 24352.571,E2 24352.571} C_VEL
LIN {X 0,Y 568.905,Z 828.798,A -85,B 0,C 180,E1 24352.279,E2 24352.279} C_VEL
LIN {X 0,Y 575.766,Z 837.975,A -85,B 0,C 180,E1 24351.402,E2 24351.402} C_VEL
LIN {X 0,Y 578.345,Z 841.639,A -85,B 0,C 180,E1 24350.91,E2 24350.91} C_VEL
LIN {X 0,Y 579.517,Z 844.823,A -85,B 0,C 180,E1 24350.308,E2 24350.308} C_VEL
LIN {X 0,Y 579.178,Z 846.904,A -85,B 0,C 180,E1 24349.733,E2 24349.733} C_VEL
LIN {X 0,Y 577.398,Z 848.22,A -85,B 0,C 180,E1 24349.114,E2 24349.114} C_VEL
LIN {X 0,Y 574.643,Z 848.504,A -85,B 0,C 180,E1 24348.583,E2 24348.583} C_VEL
LIN {X 0,Y 570.922,Z 847.81,A -85,B 0,C 180,E1 24348.099,E2 24348.099} C_VEL
LIN {X 0,Y 561.86,Z 844.1,A -85,B 0,C 180,E1 24347.153,E2 24347.153} C_VEL
LIN {X 0,Y 553.51,Z 838.63,A -85,B 0,C 180,E1 24346.116,E2 24346.116} C_VEL
LIN {X 0,Y 546.583,Z 831.833,A -85,B 0,C 180,E1 24345.067,E2 24345.067} C_VEL
LIN {X 0,Y 541.049,Z 823.784,A -85,B 0,C 180,E1 24344.015,E2 24344.015} C_VEL
LIN {X 0,Y 536.514,Z 813.512,A -85,B 0,C 180,E1 24342.861,E2 24342.861} C_VEL
LIN {X 0,Y 533.553,Z 801.619,A -85,B 0,C 180,E1 24341.702,E2 24341.702} C_VEL
LIN {X 0,Y 532.146,Z 787.162,A -85,B 0,C 180,E1 24340.452,E2 24340.452} C_VEL
LIN {X 0,Y 532.522,Z 768.499,A -85,B 0,C 180,E1 24339.038,E2 24339.038} C_VEL
LIN {X 0,Y 535.158,Z 727.748,A -85,B 0,C 180,E1 24336.052,E2 24336.052} C_VEL
LIN {X 0,Y 536,Z 714.001,A -85,B 0,C 180,E1 24335.009,E2 24335.009} C_VEL
LIN {X 0,Y 527.223,Z 697.819,A -85,B 0,C 180,E1 24332.459,E2 24332.459} C_VEL
LIN {X 0,Y 519.972,Z 684.731,A -85,B 0,C 180,E1 24330.252,E2 24330.252} C_VEL
LIN {X 0,Y 517.247,Z 679.934,A -85,B 0,C 180,E1 24329.406,E2 24329.406} C_VEL
LIN {X 0,Y 515.025,Z 675.634,A -85,B 0,C 180,E1 24328.654,E2 24328.654} C_VEL
LIN {X 0,Y 513.215,Z 673.034,A -85,B 0,C 180,E1 24328.129,E2 24328.129} C_VEL
LIN {X 0,Y 512.634,Z 670.871,A -85,B 0,C 180,E1 24327.785,E2 24327.785} C_VEL
LIN {X 0,Y 512.643,Z 670.88,A -85,B 0,C 180,E1 24324.301,E2 24324.301} C_VEL
LIN {X 0,Y 512.637,Z 670.877,A -85,B 0,C 180,E1 24320.792,E2 24320.792} C_VEL
LIN {X 0,Y 512.633,Z 670.878,A -85,B 0,C 180,E1 24317.362,E2 24317.362} C_VEL
LIN {X 0,Y 512.633,Z 670.88,A -85,B 0,C 180,E1 24313.996,E2 24313.996} C_VEL
LIN {X 0,Y 512.65,Z 670.878,A -85,B 0,C 180,E1 24310.45,E2 24310.45} C_VEL
LIN {X 0,Y 512.646,Z 670.876,A -85,B 0,C 180,E1 24306.911,E2 24306.911} C_VEL
LIN {X 0,Y 512.632,Z 670.879,A -85,B 0,C 180,E1 24303.354,E2 24303.354} C_VEL
LIN {X 0,Y 512.64,Z 670.877,A -85,B 0,C 180,E1 24299.888,E2 24299.888} C_VEL
LIN {X 0,Y 512.647,Z 670.878,A -85,B 0,C 180,E1 24296.421,E2 24296.421} C_VEL
LIN {X 0,Y 512.641,Z 670.878,A -85,B 0,C 180,E1 24292.829,E2 24292.829} C_VEL
LIN {X 0,Y 512.637,Z 670.878,A -85,B 0,C 180,E1 24289.322,E2 24289.322} C_VEL
LIN {X 0,Y 512.638,Z 670.88,A -85,B 0,C 180,E1 24285.889,E2 24285.889} C_VEL
LIN {X 0,Y 512.646,Z 670.878,A -85,B 0,C 180,E1 24282.403,E2 24282.403} C_VEL
LIN {X 0,Y 512.644,Z 670.878,A -85,B 0,C 180,E1 24278.792,E2 24278.792} C_VEL
LIN {X 0,Y 512.634,Z 670.878,A -85,B 0,C 180,E1 24275.33,E2 24275.33} C_VEL
LIN {X 0,Y 512.647,Z 670.852,A -85,B 0,C 180,E1 24271.831,E2 24271.831} C_VEL
LIN {X 0,Y 512.648,Z 670.878,A -85,B 0,C 180,E1 24268.224,E2 24268.224} C_VEL
LIN {X 0,Y 512.635,Z 670.856,A -85,B 0,C 180,E1 24264.737,E2 24264.737} C_VEL
LIN {X 0,Y 512.648,Z 670.879,A -85,B 0,C 180,E1 24261.239,E2 24261.239} C_VEL
LIN {X 0,Y 512.65,Z 670.874,A -85,B 0,C 180,E1 24257.661,E2 24257.661} C_VEL
LIN {X 0,Y 512.64,Z 670.882,A -85,B 0,C 180,E1 24254.028,E2 24254.028} C_VEL
LIN {X 0,Y 511.629,Z 671.011,A -85,B 0,C 180,E1 24253.456,E2 24253.456} C_VEL
LIN {X 0,Y 505.251,Z 671.811,A -85,B 0,C 180,E1 24251.901,E2 24251.901} C_VEL
LIN {X 0,Y 504.705,Z 671.878,A -85,B 0,C 180,E1 24251.479,E2 24251.479} C_VEL
LIN {X 0,Y 504.725,Z 672.019,A -85,B 0,C 180,E1 24251.274,E2 24251.274} C_VEL
LIN {X 0,Y 505.758,Z 674.943,A -85,B 0,C 180,E1 24250.957,E2 24250.957} C_VEL
LIN {X 0,Y 513.339,Z 691.947,A -85,B 0,C 180,E1 24248.985,E2 24248.985} C_VEL
LIN {X 0,Y 517.879,Z 703.191,A -85,B 0,C 180,E1 24247.735,E2 24247.735} C_VEL
LIN {X 0,Y 516.047,Z 749.821,A -85,B 0,C 180,E1 24244.41,E2 24244.41} C_VEL
LIN {X 0,Y 515.646,Z 768.747,A -85,B 0,C 180,E1 24243.151,E2 24243.151} C_VEL
LIN {X 0,Y 517.774,Z 783.217,A -85,B 0,C 180,E1 24242.759,E2 24242.759} C_VEL
LIN {X 0,Y 514.945,Z 1017.56,A -85,B 0,C 180,E1 24239.208,E2 24239.208} C_VEL
LIN {X 0,Y 514.454,Z 1038.972,A -85,B 0,C 180,E1 24238.782,E2 24238.782} C_VEL
LIN {X 0,Y 513.703,Z 1059.743,A -85,B 0,C 180,E1 24238.156,E2 24238.156} C_VEL
LIN {X 0,Y 512.771,Z 1079.646,A -85,B 0,C 180,E1 24237.335,E2 24237.335} C_VEL
LIN {X 0,Y 511.753,Z 1097.707,A -85,B 0,C 180,E1 24236.39,E2 24236.39} C_VEL
LIN {X 0,Y 510.603,Z 1115.836,A -85,B 0,C 180,E1 24235.219,E2 24235.219} C_VEL
LIN {X 0,Y 509.353,Z 1133.544,A -85,B 0,C 180,E1 24233.828,E2 24233.828} C_VEL
LIN {X 0,Y 508.171,Z 1150.481,A -85,B 0,C 180,E1 24232.256,E2 24232.256} C_VEL
LIN {X 0,Y 507.116,Z 1166.08,A -85,B 0,C 180,E1 24230.545,E2 24230.545} C_VEL
LIN {X 0,Y 506.179,Z 1180.622,A -85,B 0,C 180,E1 24228.662,E2 24228.662} C_VEL
LIN {X 0,Y 505.412,Z 1193.627,A -85,B 0,C 180,E1 24226.669,E2 24226.669} C_VEL
LIN {X 0,Y 504.825,Z 1205.138,A -85,B 0,C 180,E1 24224.568,E2 24224.568} C_VEL
LIN {X 0,Y 504.426,Z 1214.679,A -85,B 0,C 180,E1 24222.477,E2 24222.477} C_VEL
LIN {X 0,Y 504.145,Z 1223.221,A -85,B 0,C 180,E1 24220.166,E2 24220.166} C_VEL
LIN {X 0,Y 503.998,Z 1229.791,A -85,B 0,C 180,E1 24217.867,E2 24217.867} C_VEL
LIN {X 0,Y 503.934,Z 1234.588,A -85,B 0,C 180,E1 24215.579,E2 24215.579} C_VEL
LIN {X 0,Y 503.912,Z 1237.847,A -85,B 0,C 180,E1 24213.184,E2 24213.184} C_VEL
LIN {X 0,Y 503.911,Z 1239.341,A -85,B 0,C 180,E1 24210.795,E2 24210.795} C_VEL
LIN {X 0,Y 503.9,Z 1239.167,A -85,B 0,C 180,E1 24208.521,E2 24208.521} C_VEL
LIN {X 0,Y 503.913,Z 1237.373,A -85,B 0,C 180,E1 24206.245,E2 24206.245} C_VEL
LIN {X 0,Y 503.941,Z 1233.929,A -85,B 0,C 180,E1 24203.963,E2 24203.963} C_VEL
LIN {X 0,Y 504.007,Z 1228.819,A -85,B 0,C 180,E1 24201.673,E2 24201.673} C_VEL
LIN {X 0,Y 504.176,Z 1221.927,A -85,B 0,C 180,E1 24199.371,E2 24199.371} C_VEL
LIN {X 0,Y 504.464,Z 1213.585,A -85,B 0,C 180,E1 24197.174,E2 24197.174} C_VEL
LIN {X 0,Y 504.92,Z 1203.264,A -85,B 0,C 180,E1 24194.964,E2 24194.964} C_VEL
LIN {X 0,Y 505.575,Z 1190.922,A -85,B 0,C 180,E1 24192.788,E2 24192.788} C_VEL
LIN {X 0,Y 506.413,Z 1177.057,A -85,B 0,C 180,E1 24190.748,E2 24190.748} C_VEL
LIN {X 0,Y 507.415,Z 1161.817,A -85,B 0,C 180,E1 24188.863,E2 24188.863} C_VEL
LIN {X 0,Y 508.495,Z 1145.966,A -85,B 0,C 180,E1 24187.209,E2 24187.209} C_VEL
LIN {X 0,Y 509.757,Z 1127.916,A -85,B 0,C 180,E1 24185.613,E2 24185.613} C_VEL
LIN {X 0,Y 510.933,Z 1110.298,A -85,B 0,C 180,E1 24184.312,E2 24184.312} C_VEL
LIN {X 0,Y 512.091,Z 1091.782,A -85,B 0,C 180,E1 24183.19,E2 24183.19} C_VEL
LIN {X 0,Y 513.144,Z 1072.28,A -85,B 0,C 180,E1 24182.245,E2 24182.245} C_VEL
LIN {X 0,Y 514,Z 1052.678,A -85,B 0,C 180,E1 24181.513,E2 24181.513} C_VEL
LIN {X 0,Y 514.668,Z 1032.125,A -85,B 0,C 180,E1 24180.964,E2 24180.964} C_VEL
LIN {X 0,Y 515.141,Z 1000.234,A -85,B 0,C 180,E1 24180.442,E2 24180.442} C_VEL
LIN {X 0,Y 517.662,Z 787.549,A -85,B 0,C 180,E1 24177.213,E2 24177.213} C_VEL
LIN {X 0,Y 513.575,Z 769.698,A -85,B 0,C 180,E1 24176.599,E2 24176.599} C_VEL
LIN {X 0,Y 514.761,Z 735.945,A -85,B 0,C 180,E1 24173.255,E2 24173.255} C_VEL
LIN {X 0,Y 516.259,Z 703.032,A -85,B 0,C 180,E1 24169.817,E2 24169.817} C_VEL
LIN {X 0,Y 509.945,Z 685.4,A -85,B 0,C 180,E1 24167.33,E2 24167.33} C_VEL
LIN {X 0,Y 504.695,Z 671.868,A -85,B 0,C 180,E1 24165.396,E2 24165.396} C_VEL
LIN {X 0,Y 504.708,Z 671.869,A -85,B 0,C 180,E1 24161.851,E2 24161.851} C_VEL
LIN {X 0,Y 504.71,Z 671.918,A -85,B 0,C 180,E1 24158.412,E2 24158.412} C_VEL
LIN {X 0,Y 513.185,Z 693.127,A -85,B 0,C 180,E1 24155.471,E2 24155.471} C_VEL
LIN {X 0,Y 516.486,Z 702.23,A -85,B 0,C 180,E1 24154.288,E2 24154.288} C_VEL
LIN {X 0,Y 514.476,Z 739.154,A -85,B 0,C 180,E1 24150.934,E2 24150.934} C_VEL
LIN {X 0,Y 512.437,Z 778.5,A -85,B 0,C 180,E1 24147.418,E2 24147.418} C_VEL
LIN {X 0,Y 510.506,Z 818.997,A -85,B 0,C 180,E1 24143.844,E2 24143.844} C_VEL
LIN {X 0,Y 509.302,Z 848.28,A -85,B 0,C 180,E1 24141.314,E2 24141.314} C_VEL
LIN {X 0,Y 510.497,Z 858.739,A -85,B 0,C 180,E1 24141.071,E2 24141.071} C_VEL
LIN {X 0,Y 508.962,Z 1013.813,A -85,B 0,C 180,E1 24138.732,E2 24138.732} C_VEL
LIN {X 0,Y 508.663,Z 1029.507,A -85,B 0,C 180,E1 24138.357,E2 24138.357} C_VEL
LIN {X 0,Y 508.227,Z 1046.307,A -85,B 0,C 180,E1 24137.755,E2 24137.755} C_VEL
LIN {X 0,Y 507.677,Z 1061.185,A -85,B 0,C 180,E1 24137.016,E2 24137.016} C_VEL
LIN {X 0,Y 507.122,Z 1074.207,A -85,B 0,C 180,E1 24136.206,E2 24136.206} C_VEL
LIN {X 0,Y 506.55,Z 1086.444,A -85,B 0,C 180,E1 24135.279,E2 24135.279} C_VEL
LIN {X 0,Y 505.929,Z 1099.666,A -85,B 0,C 180,E1 24134.069,E2 24134.069} C_VEL
LIN {X 0,Y 505.314,Z 1111.789,A -85,B 0,C 180,E1 24132.688,E2 24132.688} C_VEL
LIN {X 0,Y 504.821,Z 1122.721,A -85,B 0,C 180,E1 24131.192,E2 24131.192} C_VEL
LIN {X 0,Y 504.457,Z 1132.609,A -85,B 0,C 180,E1 24129.584,E2 24129.584} C_VEL
LIN {X 0,Y 504.176,Z 1141.453,A -85,B 0,C 180,E1 24127.75,E2 24127.75} C_VEL
LIN {X 0,Y 504.044,Z 1147.191,A -85,B 0,C 180,E1 24126.264,E2 24126.264} C_VEL
LIN {X 0,Y 503.967,Z 1151.735,A -85,B 0,C 180,E1 24124.78,E2 24124.78} C_VEL
LIN {X 0,Y 503.927,Z 1155.406,A -85,B 0,C 180,E1 24123.185,E2 24123.185} C_VEL
LIN {X 0,Y 503.914,Z 1158.322,A -85,B 0,C 180,E1 24121.251,E2 24121.251} C_VEL
LIN {X 0,Y 503.915,Z 1159.408,A -85,B 0,C 180,E1 24119.204,E2 24119.204} C_VEL
LIN {X 0,Y 503.915,Z 1158.935,A -85,B 0,C 180,E1 24117.498,E2 24117.498} C_VEL
LIN {X 0,Y 503.917,Z 1157.334,A -85,B 0,C 180,E1 24115.904,E2 24115.904} C_VEL
LIN {X 0,Y 503.941,Z 1154.121,A -85,B 0,C 180,E1 24114.078,E2 24114.078} C_VEL
LIN {X 0,Y 504.013,Z 1148.848,A -85,B 0,C 180,E1 24112.133,E2 24112.133} C_VEL
LIN {X 0,Y 504.14,Z 1142.978,A -85,B 0,C 180,E1 24110.525,E2 24110.525} C_VEL
LIN {X 0,Y 504.332,Z 1136.186,A -85,B 0,C 180,E1 24109.029,E2 24109.029} C_VEL
LIN {X 0,Y 504.619,Z 1127.925,A -85,B 0,C 180,E1 24107.528,E2 24107.528} C_VEL
LIN {X 0,Y 505.154,Z 1115.427,A -85,B 0,C 180,E1 24105.676,E2 24105.676} C_VEL
LIN {X 0,Y 505.661,Z 1105.588,A -85,B 0,C 180,E1 24104.459,E2 24104.459} C_VEL
LIN {X 0,Y 506.249,Z 1094.575,A -85,B 0,C 180,E1 24103.314,E2 24103.314} C_VEL
LIN {X 0,Y 506.945,Z 1081,A -85,B 0,C 180,E1 24102.147,E2 24102.147} C_VEL
LIN {X 0,Y 507.621,Z 1065.363,A -85,B 0,C 180,E1 24101.094,E2 24101.094} C_VEL
LIN {X 0,Y 508.155,Z 1050.99,A -85,B 0,C 180,E1 24100.339,E2 24100.339} C_VEL
LIN {X 0,Y 508.648,Z 1034.47,A -85,B 0,C 180,E1 24099.683,E2 24099.683} C_VEL
LIN {X 0,Y 508.938,Z 1017.283,A -85,B 0,C 180,E1 24099.238,E2 24099.238} C_VEL
LIN {X 0,Y 510.713,Z 880.716,A -85,B 0,C 180,E1 24097.065,E2 24097.065} C_VEL
LIN {X 0,Y 511.002,Z 855.753,A -85,B 0,C 180,E1 24096.627,E2 24096.627} C_VEL
LIN {X 0,Y 511.728,Z 849.756,A -85,B 0,C 180,E1 24096.124,E2 24096.124} C_VEL
LIN {X 0,Y 515.128,Z 816.687,A -85,B 0,C 180,E1 24092.862,E2 24092.862} C_VEL
LIN {X 0,Y 519.2,Z 789.454,A -85,B 0,C 180,E1 24090.018,E2 24090.018} C_VEL
LIN {X 0,Y 524.168,Z 766.661,A -85,B 0,C 180,E1 24087.458,E2 24087.458} C_VEL
LIN {X 0,Y 529.927,Z 748.667,A -85,B 0,C 180,E1 24085.263,E2 24085.263} C_VEL
LIN {X 0,Y 535.608,Z 736.403,A -85,B 0,C 180,E1 24083.593,E2 24083.593} C_VEL
LIN {X 0,Y 527.86,Z 748.111,A -85,B 0,C 180,E1 24082.351,E2 24082.351} C_VEL
LIN {X 0,Y 522.514,Z 759.962,A -85,B 0,C 180,E1 24081.153,E2 24081.153} C_VEL
LIN {X 0,Y 519.412,Z 772.059,A -85,B 0,C 180,E1 24079.989,E2 24079.989} C_VEL
LIN {X 0,Y 518.36,Z 785.059,A -85,B 0,C 180,E1 24078.787,E2 24078.787} C_VEL
LIN {X 0,Y 519.452,Z 797.55,A -85,B 0,C 180,E1 24077.648,E2 24077.648} C_VEL
LIN {X 0,Y 522.575,Z 809.622,A -85,B 0,C 180,E1 24076.541,E2 24076.541} C_VEL
LIN {X 0,Y 527.382,Z 820.399,A -85,B 0,C 180,E1 24075.531,E2 24075.531} C_VEL
LIN {X 0,Y 533.684,Z 829.928,A -85,B 0,C 180,E1 24074.608,E2 24074.608} C_VEL
LIN {X 0,Y 541.319,Z 838.343,A -85,B 0,C 180,E1 24073.763,E2 24073.763} C_VEL
LIN {X 0,Y 551.417,Z 846.499,A -85,B 0,C 180,E1 24072.899,E2 24072.899} C_VEL
LIN {X 0,Y 562.313,Z 852.807,A -85,B 0,C 180,E1 24072.143,E2 24072.143} C_VEL
LIN {X 0,Y 567.076,Z 854.704,A -85,B 0,C 180,E1 24071.77,E2 24071.77} C_VEL
LIN {X 0,Y 571.688,Z 855.699,A -85,B 0,C 180,E1 24071.232,E2 24071.232} C_VEL
LIN {X 0,Y 574.805,Z 855.482,A -85,B 0,C 180,E1 24070.676,E2 24070.676} C_VEL
LIN {X 0,Y 576.629,Z 854.41,A -85,B 0,C 180,E1 24070.122,E2 24070.122} C_VEL
LIN {X 0,Y 577.264,Z 852.203,A -85,B 0,C 180,E1 24069.47,E2 24069.47} C_VEL
LIN {X 0,Y 576.289,Z 849.188,A -85,B 0,C 180,E1 24068.873,E2 24068.873} C_VEL
LIN {X 0,Y 573.735,Z 845.478,A -85,B 0,C 180,E1 24068.346,E2 24068.346} C_VEL
LIN {X 0,Y 572.157,Z 843.917,A -85,B 0,C 180,E1 24068.14,E2 24068.14} C_VEL
LIN {X 0,Y 568.488,Z 869.068,A -85,B 0,C 180,E1 24067.739,E2 24067.739} C_VEL
LIN {X 0,Y 565.288,Z 883.446,A -85,B 0,C 180,E1 24067.414,E2 24067.414} C_VEL
LIN {X 0,Y 564.14,Z 888.01,A -85,B 0,C 180,E1 24067.289,E2 24067.289} C_VEL
LIN {X 0,Y 559.577,Z 909.268,A -85,B 0,C 180,E1 24067.188,E2 24067.188} C_VEL
LIN {X 0,Y 553.003,Z 930.54,A -85,B 0,C 180,E1 24067.069,E2 24067.069} C_VEL
LIN {X 0,Y 545.466,Z 950.086,A -85,B 0,C 180,E1 24066.86,E2 24066.86} C_VEL
LIN {X 0,Y 539.264,Z 965.6,A -85,B 0,C 180,E1 24066.525,E2 24066.525} C_VEL
LIN {X 0,Y 535.585,Z 976.292,A -85,B 0,C 180,E1 24066.152,E2 24066.152} C_VEL
LIN {X 0,Y 534.185,Z 979.971,A -85,B 0,C 180,E1 24066.042,E2 24066.042} C_VEL
LIN {X 0,Y 528.755,Z 992.987,A -85,B 0,C 180,E1 24065.688,E2 24065.688} C_VEL
LIN {X 0,Y 525.109,Z 1004.229,A -85,B 0,C 180,E1 24065.236,E2 24065.236} C_VEL
LIN {X 0,Y 520.886,Z 1017.463,A -85,B 0,C 180,E1 24064.691,E2 24064.691} C_VEL
LIN {X 0,Y 519,Z 1025.319,A -85,B 0,C 180,E1 24064.343,E2 24064.343} C_VEL
LIN {X 0,Y 518.301,Z 1067.056,A -85,B 0,C 180,E1 24063.664,E2 24063.664} C_VEL
LIN {X 0,Y 517.475,Z 1089.094,A -85,B 0,C 180,E1 24063.107,E2 24063.107} C_VEL
LIN {X 0,Y 516.433,Z 1111.049,A -85,B 0,C 180,E1 24062.334,E2 24062.334} C_VEL
LIN {X 0,Y 515.223,Z 1131.649,A -85,B 0,C 180,E1 24061.397,E2 24061.397} C_VEL
LIN {X 0,Y 513.826,Z 1152.277,A -85,B 0,C 180,E1 24060.234,E2 24060.234} C_VEL
LIN {X 0,Y 512.35,Z 1172.121,A -85,B 0,C 180,E1 24058.872,E2 24058.872} C_VEL
LIN {X 0,Y 510.816,Z 1191.804,A -85,B 0,C 180,E1 24057.26,E2 24057.26} C_VEL
LIN {X 0,Y 509.45,Z 1208.579,A -85,B 0,C 180,E1 24055.643,E2 24055.643} C_VEL
LIN {X 0,Y 508.315,Z 1223.155,A -85,B 0,C 180,E1 24054.028,E2 24054.028} C_VEL
LIN {X 0,Y 507.131,Z 1239.061,A -85,B 0,C 180,E1 24052,E2 24052} C_VEL
LIN {X 0,Y 506.134,Z 1253.09,A -85,B 0,C 180,E1 24049.894,E2 24049.894} C_VEL
LIN {X 0,Y 505.403,Z 1264.822,A -85,B 0,C 180,E1 24047.857,E2 24047.857} C_VEL
LIN {X 0,Y 504.759,Z 1276.831,A -85,B 0,C 180,E1 24045.393,E2 24045.393} C_VEL
LIN {X 0,Y 504.381,Z 1285.797,A -85,B 0,C 180,E1 24043.178,E2 24043.178} C_VEL
LIN {X 0,Y 504.132,Z 1293.556,A -85,B 0,C 180,E1 24040.861,E2 24040.861} C_VEL
LIN {X 0,Y 503.981,Z 1300.14,A -85,B 0,C 180,E1 24038.328,E2 24038.328} C_VEL
LIN {X 0,Y 503.922,Z 1304.392,A -85,B 0,C 180,E1 24036.151,E2 24036.151} C_VEL
LIN {X 0,Y 503.9,Z 1307.596,A -85,B 0,C 180,E1 24033.755,E2 24033.755} C_VEL
LIN {X 0,Y 503.906,Z 1309.235,A -85,B 0,C 180,E1 24031.251,E2 24031.251} C_VEL
LIN {X 0,Y 503.905,Z 1309.316,A -85,B 0,C 180,E1 24029.091,E2 24029.091} C_VEL
LIN {X 0,Y 503.912,Z 1307.935,A -85,B 0,C 180,E1 24026.588,E2 24026.588} C_VEL
LIN {X 0,Y 503.923,Z 1304.783,A -85,B 0,C 180,E1 24024.078,E2 24024.078} C_VEL
LIN {X 0,Y 503.981,Z 1300.584,A -85,B 0,C 180,E1 24021.879,E2 24021.879} C_VEL
LIN {X 0,Y 504.098,Z 1295.078,A -85,B 0,C 180,E1 24019.67,E2 24019.67} C_VEL
LIN {X 0,Y 504.349,Z 1286.68,A -85,B 0,C 180,E1 24017.055,E2 24017.055} C_VEL
LIN {X 0,Y 504.731,Z 1277.329,A -85,B 0,C 180,E1 24014.725,E2 24014.725} C_VEL
LIN {X 0,Y 505.333,Z 1266.119,A -85,B 0,C 180,E1 24012.379,E2 24012.379} C_VEL
LIN {X 0,Y 506.077,Z 1254.014,A -85,B 0,C 180,E1 24010.255,E2 24010.255} C_VEL
LIN {X 0,Y 506.999,Z 1240.739,A -85,B 0,C 180,E1 24008.238,E2 24008.238} C_VEL
LIN {X 0,Y 508.241,Z 1224.192,A -85,B 0,C 180,E1 24006.093,E2 24006.093} C_VEL
LIN {X 0,Y 509.405,Z 1209.163,A -85,B 0,C 180,E1 24004.418,E2 24004.418} C_VEL
LIN {X 0,Y 510.762,Z 1192.491,A -85,B 0,C 180,E1 24002.801,E2 24002.801} C_VEL
LIN {X 0,Y 512.292,Z 1172.796,A -85,B 0,C 180,E1 24001.18,E2 24001.18} C_VEL
LIN {X 0,Y 513.788,Z 1152.784,A -85,B 0,C 180,E1 23999.798,E2 23999.798} C_VEL
LIN {X 0,Y 515.17,Z 1132.509,A -85,B 0,C 180,E1 23998.645,E2 23998.645} C_VEL
LIN {X 0,Y 516.395,Z 1111.836,A -85,B 0,C 180,E1 23997.698,E2 23997.698} C_VEL
LIN {X 0,Y 517.433,Z 1090.003,A -85,B 0,C 180,E1 23996.92,E2 23996.92} C_VEL
LIN {X 0,Y 518.282,Z 1067.636,A -85,B 0,C 180,E1 23996.348,E2 23996.348} C_VEL
LIN {X 0,Y 518.949,Z 1029.166,A -85,B 0,C 180,E1 23995.716,E2 23995.716} C_VEL
LIN {X 0,Y 519.042,Z 1024.446,A -85,B 0,C 180,E1 23995.639,E2 23995.639} C_VEL
LIN {X 0,Y 523.317,Z 1009.403,A -85,B 0,C 180,E1 23994.961,E2 23994.961} C_VEL
LIN {X 0,Y 525.649,Z 1002.256,A -85,B 0,C 180,E1 23994.673,E2 23994.673} C_VEL
LIN {X 0,Y 529.566,Z 990.879,A -85,B 0,C 180,E1 23994.243,E2 23994.243} C_VEL
LIN {X 0,Y 535.291,Z 977.306,A -85,B 0,C 180,E1 23993.892,E2 23993.892} C_VEL
LIN {X 0,Y 538.831,Z 966.747,A -85,B 0,C 180,E1 23993.508,E2 23993.508} C_VEL
LIN {X 0,Y 545.179,Z 950.793,A -85,B 0,C 180,E1 23993.151,E2 23993.151} C_VEL
LIN {X 0,Y 552.546,Z 931.82,A -85,B 0,C 180,E1 23992.94,E2 23992.94} C_VEL
LIN {X 0,Y 559.347,Z 910.136,A -85,B 0,C 180,E1 23992.816,E2 23992.816} C_VEL
LIN {X 0,Y 563.975,Z 888.983,A -85,B 0,C 180,E1 23992.716,E2 23992.716} C_VEL
LIN {X 0,Y 564.641,Z 885.803,A -85,B 0,C 180,E1 23992.664,E2 23992.664} C_VEL
LIN {X 0,Y 567.604,Z 873.528,A -85,B 0,C 180,E1 23992.344,E2 23992.344} C_VEL
LIN {X 0,Y 571.321,Z 850.859,A -85,B 0,C 180,E1 23991.966,E2 23991.966} C_VEL
LIN {X 0,Y 572.209,Z 843.691,A -85,B 0,C 180,E1 23991.853,E2 23991.853} C_VEL
LIN {X 0,Y 575.464,Z 847.8,A -85,B 0,C 180,E1 23991.346,E2 23991.346} C_VEL
LIN {X 0,Y 577.069,Z 851.1,A -85,B 0,C 180,E1 23990.772,E2 23990.772} C_VEL
LIN {X 0,Y 577.072,Z 853.667,A -85,B 0,C 180,E1 23990.135,E2 23990.135} C_VEL
LIN {X 0,Y 575.635,Z 855.17,A -85,B 0,C 180,E1 23989.534,E2 23989.534} C_VEL
LIN {X 0,Y 572.816,Z 855.753,A -85,B 0,C 180,E1 23988.943,E2 23988.943} C_VEL
LIN {X 0,Y 569.172,Z 855.292,A -85,B 0,C 180,E1 23988.447,E2 23988.447} C_VEL
LIN {X 0,Y 559.303,Z 851.662,A -85,B 0,C 180,E1 23987.436,E2 23987.436} C_VEL
LIN {X 0,Y 550.757,Z 846.59,A -85,B 0,C 180,E1 23986.415,E2 23986.415} C_VEL
LIN {X 0,Y 543.007,Z 839.766,A -85,B 0,C 180,E1 23985.296,E2 23985.296} C_VEL
LIN {X 0,Y 536.728,Z 831.595,A -85,B 0,C 180,E1 23984.164,E2 23984.164} C_VEL
LIN {X 0,Y 531.806,Z 821.81,A -85,B 0,C 180,E1 23983,E2 23983} C_VEL
LIN {X 0,Y 528.189,Z 809.9,A -85,B 0,C 180,E1 23981.77,E2 23981.77} C_VEL
LIN {X 0,Y 526.257,Z 796.273,A -85,B 0,C 180,E1 23980.525,E2 23980.525} C_VEL
LIN {X 0,Y 525.966,Z 779.772,A -85,B 0,C 180,E1 23979.196,E2 23979.196} C_VEL
LIN {X 0,Y 529.147,Z 731.865,A -85,B 0,C 180,E1 23975.659,E2 23975.659} C_VEL
LIN {X 0,Y 529.96,Z 718.269,A -85,B 0,C 180,E1 23974.603,E2 23974.603} C_VEL
LIN {X 0,Y 519.984,Z 699.947,A -85,B 0,C 180,E1 23971.664,E2 23971.664} C_VEL
LIN {X 0,Y 514.478,Z 690.112,A -85,B 0,C 180,E1 23969.964,E2 23969.964} C_VEL
LIN {X 0,Y 512.144,Z 685.865,A -85,B 0,C 180,E1 23969.214,E2 23969.214} C_VEL
LIN {X 0,Y 509.48,Z 681.141,A -85,B 0,C 180,E1 23968.354,E2 23968.354} C_VEL
LIN {X 0,Y 507.565,Z 677.529,A -85,B 0,C 180,E1 23967.703,E2 23967.703} C_VEL
LIN {X 0,Y 505.194,Z 673.803,A -85,B 0,C 180,E1 23966.951,E2 23966.951} C_VEL
LIN {X 0,Y 504.701,Z 671.857,A -85,B 0,C 180,E1 23966.647,E2 23966.647} C_VEL
LIN {X 0,Y 504.708,Z 671.865,A -85,B 0,C 180,E1 23963.094,E2 23963.094} C_VEL
LIN {X 0,Y 504.703,Z 671.869,A -85,B 0,C 180,E1 23959.56,E2 23959.56} C_VEL
LIN {X 0,Y 504.699,Z 671.868,A -85,B 0,C 180,E1 23956.092,E2 23956.092} C_VEL
LIN {X 0,Y 504.7,Z 671.868,A -85,B 0,C 180,E1 23952.587,E2 23952.587} C_VEL
LIN {X 0,Y 504.712,Z 671.869,A -85,B 0,C 180,E1 23949.004,E2 23949.004} C_VEL
LIN {X 0,Y 504.703,Z 671.869,A -85,B 0,C 180,E1 23945.57,E2 23945.57} C_VEL
LIN {X 0,Y 504.694,Z 671.867,A -85,B 0,C 180,E1 23942.043,E2 23942.043} C_VEL
LIN {X 0,Y 504.703,Z 671.867,A -85,B 0,C 180,E1 23938.524,E2 23938.524} C_VEL
LIN {X 0,Y 504.71,Z 671.87,A -85,B 0,C 180,E1 23934.999,E2 23934.999} C_VEL
LIN {X 0,Y 504.693,Z 671.867,A -85,B 0,C 180,E1 23931.455,E2 23931.455} C_VEL
LIN {X 0,Y 504.694,Z 671.868,A -85,B 0,C 180,E1 23927.994,E2 23927.994} C_VEL
LIN {X 0,Y 504.705,Z 671.868,A -85,B 0,C 180,E1 23924.487,E2 23924.487} C_VEL
LIN {X 0,Y 504.704,Z 671.861,A -85,B 0,C 180,E1 23921.04,E2 23921.04} C_VEL
LIN {X 0,Y 504.696,Z 671.864,A -85,B 0,C 180,E1 23917.643,E2 23917.643} C_VEL
LIN {X 0,Y 504.693,Z 671.867,A -85,B 0,C 180,E1 23914.161,E2 23914.161} C_VEL
LIN {X 0,Y 504.694,Z 671.838,A -85,B 0,C 180,E1 23910.703,E2 23910.703} C_VEL
LIN {X 0,Y 504.71,Z 671.868,A -85,B 0,C 180,E1 23907.26,E2 23907.26} C_VEL
LIN {X 0,Y 504.698,Z 671.85,A -85,B 0,C 180,E1 23903.676,E2 23903.676} C_VEL
LIN {X 0,Y 504.692,Z 671.858,A -85,B 0,C 180,E1 23900.215,E2 23900.215} C_VEL
LIN {X 0,Y 504.699,Z 671.87,A -85,B 0,C 180,E1 23896.728,E2 23896.728} C_VEL
LIN {X 0,Y 504.71,Z 671.874,A -85,B 0,C 180,E1 23893.195,E2 23893.195} C_VEL
LIN {X 0,Y 504.705,Z 671.878,A -85,B 0,C 180,E1 23891.479,E2 23891.479} C_VEL
LIN {X 0,Y 505.701,Z 672.496,A -85,B 0,C 180,E1 23891.16,E2 23891.16} C_VEL
LIN {X 0,Y 508.121,Z 675.307,A -85,B 0,C 180,E1 23890.716,E2 23890.716} C_VEL
LIN {X 0,Y 509.083,Z 679.52,A -85,B 0,C 180,E1 23890.312,E2 23890.312} C_VEL
LIN {X 0,Y 509.073,Z 685.703,A -85,B 0,C 180,E1 23889.89,E2 23889.89} C_VEL
LIN {X 0,Y 507.599,Z 695.288,A -85,B 0,C 180,E1 23889.249,E2 23889.249} C_VEL
LIN {X 0,Y 508.077,Z 699.007,A -85,B 0,C 180,E1 23888.898,E2 23888.898} C_VEL
LIN {X 0,Y 511.039,Z 706.696,A -85,B 0,C 180,E1 23888.046,E2 23888.046} C_VEL
LIN {X 0,Y 509.144,Z 752.029,A -85,B 0,C 180,E1 23884.79,E2 23884.79} C_VEL
LIN {X 0,Y 508.793,Z 769.069,A -85,B 0,C 180,E1 23883.66,E2 23883.66} C_VEL
LIN {X 0,Y 511.067,Z 784.603,A -85,B 0,C 180,E1 23883.23,E2 23883.23} C_VEL
LIN {X 0,Y 507.966,Z 1019.607,A -85,B 0,C 180,E1 23879.623,E2 23879.623} C_VEL
LIN {X 0,Y 507.449,Z 1040.423,A -85,B 0,C 180,E1 23879.193,E2 23879.193} C_VEL
LIN {X 0,Y 506.65,Z 1060.845,A -85,B 0,C 180,E1 23878.562,E2 23878.562} C_VEL
LIN {X 0,Y 505.68,Z 1080.221,A -85,B 0,C 180,E1 23877.751,E2 23877.751} C_VEL
LIN {X 0,Y 504.591,Z 1098.294,A -85,B 0,C 180,E1 23876.794,E2 23876.794} C_VEL
LIN {X 0,Y 503.339,Z 1116.59,A -85,B 0,C 180,E1 23875.597,E2 23875.597} C_VEL
LIN {X 0,Y 501.984,Z 1134.363,A -85,B 0,C 180,E1 23874.181,E2 23874.181} C_VEL
LIN {X 0,Y 500.722,Z 1150.24,A -85,B 0,C 180,E1 23872.667,E2 23872.667} C_VEL
LIN {X 0,Y 499.505,Z 1165.604,A -85,B 0,C 180,E1 23870.934,E2 23870.934} C_VEL
LIN {X 0,Y 498.434,Z 1180.625,A -85,B 0,C 180,E1 23868.963,E2 23868.963} C_VEL
LIN {X 0,Y 497.584,Z 1193.629,A -85,B 0,C 180,E1 23866.939,E2 23866.939} C_VEL
LIN {X 0,Y 496.933,Z 1205.14,A -85,B 0,C 180,E1 23864.804,E2 23864.804} C_VEL
LIN {X 0,Y 496.487,Z 1214.684,A -85,B 0,C 180,E1 23862.68,E2 23862.68} C_VEL
LIN {X 0,Y 496.172,Z 1223.223,A -85,B 0,C 180,E1 23860.331,E2 23860.331} C_VEL
LIN {X 0,Y 496.006,Z 1229.793,A -85,B 0,C 180,E1 23857.995,E2 23857.995} C_VEL
LIN {X 0,Y 495.939,Z 1234.59,A -85,B 0,C 180,E1 23855.669,E2 23855.669} C_VEL
LIN {X 0,Y 495.912,Z 1237.735,A -85,B 0,C 180,E1 23853.351,E2 23853.351} C_VEL
LIN {X 0,Y 495.913,Z 1239.296,A -85,B 0,C 180,E1 23851.039,E2 23851.039} C_VEL
LIN {X 0,Y 495.905,Z 1239.269,A -85,B 0,C 180,E1 23848.729,E2 23848.729} C_VEL
LIN {X 0,Y 495.912,Z 1237.579,A -85,B 0,C 180,E1 23846.397,E2 23846.397} C_VEL
LIN {X 0,Y 495.941,Z 1234.337,A -85,B 0,C 180,E1 23844.098,E2 23844.098} C_VEL
LIN {X 0,Y 496.01,Z 1229.418,A -85,B 0,C 180,E1 23841.771,E2 23841.771} C_VEL
LIN {X 0,Y 496.173,Z 1223.101,A -85,B 0,C 180,E1 23839.543,E2 23839.543} C_VEL
LIN {X 0,Y 496.493,Z 1214.569,A -85,B 0,C 180,E1 23837.201,E2 23837.201} C_VEL
LIN {X 0,Y 496.974,Z 1204.406,A -85,B 0,C 180,E1 23834.953,E2 23834.953} C_VEL
LIN {X 0,Y 497.64,Z 1192.753,A -85,B 0,C 180,E1 23832.821,E2 23832.821} C_VEL
LIN {X 0,Y 498.468,Z 1180.074,A -85,B 0,C 180,E1 23830.868,E2 23830.868} C_VEL
LIN {X 0,Y 499.564,Z 1164.847,A -85,B 0,C 180,E1 23828.883,E2 23828.883} C_VEL
LIN {X 0,Y 500.793,Z 1149.339,A -85,B 0,C 180,E1 23827.151,E2 23827.151} C_VEL
LIN {X 0,Y 502.097,Z 1132.761,A -85,B 0,C 180,E1 23825.593,E2 23825.593} C_VEL
LIN {X 0,Y 503.368,Z 1116.082,A -85,B 0,C 180,E1 23824.277,E2 23824.277} C_VEL
LIN {X 0,Y 504.642,Z 1097.633,A -85,B 0,C 180,E1 23823.075,E2 23823.075} C_VEL
LIN {X 0,Y 505.759,Z 1078.844,A -85,B 0,C 180,E1 23822.092,E2 23822.092} C_VEL
LIN {X 0,Y 506.725,Z 1059.274,A -85,B 0,C 180,E1 23821.292,E2 23821.292} C_VEL
LIN {X 0,Y 507.491,Z 1038.531,A -85,B 0,C 180,E1 23820.669,E2 23820.669} C_VEL
LIN {X 0,Y 508.021,Z 1015.263,A -85,B 0,C 180,E1 23820.22,E2 23820.22} C_VEL
LIN {X 0,Y 510.977,Z 789.262,A -85,B 0,C 180,E1 23816.751,E2 23816.751} C_VEL
LIN {X 0,Y 506.587,Z 770.152,A -85,B 0,C 180,E1 23816.084,E2 23816.084} C_VEL
LIN {X 0,Y 507.748,Z 738.092,A -85,B 0,C 180,E1 23812.895,E2 23812.895} C_VEL
LIN {X 0,Y 509.294,Z 706.447,A -85,B 0,C 180,E1 23809.563,E2 23809.563} C_VEL
LIN {X 0,Y 503.313,Z 689.59,A -85,B 0,C 180,E1 23807.142,E2 23807.142} C_VEL
LIN {X 0,Y 497.847,Z 676.003,A -85,B 0,C 180,E1 23805.15,E2 23805.15} C_VEL
LIN {X 0,Y 496.768,Z 672.858,A -85,B 0,C 180,E1 23804.691,E2 23804.691} C_VEL
LIN {X 0,Y 496.756,Z 672.851,A -85,B 0,C 180,E1 23801.161,E2 23801.161} C_VEL
LIN {X 0,Y 496.795,Z 673.091,A -85,B 0,C 180,E1 23799.116,E2 23799.116} C_VEL
LIN {X 0,Y 498.251,Z 676.607,A -85,B 0,C 180,E1 23798.599,E2 23798.599} C_VEL
LIN {X 0,Y 506.4,Z 696.71,A -85,B 0,C 180,E1 23795.757,E2 23795.757} C_VEL
LIN {X 0,Y 509.586,Z 705.26,A -85,B 0,C 180,E1 23794.613,E2 23794.613} C_VEL
LIN {X 0,Y 507.545,Z 740.963,A -85,B 0,C 180,E1 23791.338,E2 23791.338} C_VEL
LIN {X 0,Y 505.39,Z 779.849,A -85,B 0,C 180,E1 23787.829,E2 23787.829} C_VEL
LIN {X 0,Y 503.305,Z 821.121,A -85,B 0,C 180,E1 23784.157,E2 23784.157} C_VEL
LIN {X 0,Y 502.063,Z 849.293,A -85,B 0,C 180,E1 23781.699,E2 23781.699} C_VEL
LIN {X 0,Y 503.271,Z 859.721,A -85,B 0,C 180,E1 23781.449,E2 23781.449} C_VEL
LIN {X 0,Y 501.452,Z 1015.747,A -85,B 0,C 180,E1 23779.019,E2 23779.019} C_VEL
LIN {X 0,Y 501.127,Z 1032.582,A -85,B 0,C 180,E1 23778.594,E2 23778.594} C_VEL
LIN {X 0,Y 500.595,Z 1050.059,A -85,B 0,C 180,E1 23777.914,E2 23777.914} C_VEL
LIN {X 0,Y 500.022,Z 1064.6,A -85,B 0,C 180,E1 23777.155,E2 23777.155} C_VEL
LIN {X 0,Y 499.338,Z 1079.63,A -85,B 0,C 180,E1 23776.161,E2 23776.161} C_VEL
LIN {X 0,Y 498.597,Z 1094.245,A -85,B 0,C 180,E1 23774.933,E2 23774.933} C_VEL
LIN {X 0,Y 497.958,Z 1106.143,A -85,B 0,C 180,E1 23773.706,E2 23773.706} C_VEL
LIN {X 0,Y 497.412,Z 1116.556,A -85,B 0,C 180,E1 23772.421,E2 23772.421} C_VEL
LIN {X 0,Y 496.859,Z 1127.498,A -85,B 0,C 180,E1 23770.787,E2 23770.787} C_VEL
LIN {X 0,Y 496.452,Z 1136.199,A -85,B 0,C 180,E1 23769.155,E2 23769.155} C_VEL
LIN {X 0,Y 496.199,Z 1142.79,A -85,B 0,C 180,E1 23767.643,E2 23767.643} C_VEL
LIN {X 0,Y 496.037,Z 1148.474,A -85,B 0,C 180,E1 23766.017,E2 23766.017} C_VEL
LIN {X 0,Y 495.942,Z 1154.3,A -85,B 0,C 180,E1 23763.815,E2 23763.815} C_VEL
LIN {X 0,Y 495.917,Z 1157.296,A -85,B 0,C 180,E1 23762.08,E2 23762.08} C_VEL
LIN {X 0,Y 495.915,Z 1158.912,A -85,B 0,C 180,E1 23760.462,E2 23760.462} C_VEL
LIN {X 0,Y 495.914,Z 1159.401,A -85,B 0,C 180,E1 23758.845,E2 23758.845} C_VEL
LIN {X 0,Y 495.915,Z 1158.695,A -85,B 0,C 180,E1 23757.111,E2 23757.111} C_VEL
LIN {X 0,Y 495.925,Z 1156.123,A -85,B 0,C 180,E1 23755.027,E2 23755.027} C_VEL
LIN {X 0,Y 495.966,Z 1152.388,A -85,B 0,C 180,E1 23753.285,E2 23753.285} C_VEL
LIN {X 0,Y 496.08,Z 1147.077,A -85,B 0,C 180,E1 23751.423,E2 23751.423} C_VEL
LIN {X 0,Y 496.335,Z 1140.162,A -85,B 0,C 180,E1 23749.555,E2 23749.555} C_VEL
LIN {X 0,Y 496.727,Z 1131.634,A -85,B 0,C 180,E1 23747.799,E2 23747.799} C_VEL
LIN {X 0,Y 497.224,Z 1122.568,A -85,B 0,C 180,E1 23746.274,E2 23746.274} C_VEL
LIN {X 0,Y 497.835,Z 1111.515,A -85,B 0,C 180,E1 23744.746,E2 23744.746} C_VEL
LIN {X 0,Y 498.575,Z 1098.426,A -85,B 0,C 180,E1 23743.293,E2 23743.293} C_VEL
LIN {X 0,Y 499.246,Z 1085.845,A -85,B 0,C 180,E1 23742.157,E2 23742.157} C_VEL
LIN {X 0,Y 499.974,Z 1071.015,A -85,B 0,C 180,E1 23741.071,E2 23741.071} C_VEL
LIN {X 0,Y 500.585,Z 1055.218,A -85,B 0,C 180,E1 23740.181,E2 23740.181} C_VEL
LIN {X 0,Y 501.089,Z 1038.795,A -85,B 0,C 180,E1 23739.49,E2 23739.49} C_VEL
LIN {X 0,Y 501.426,Z 1021.289,A -85,B 0,C 180,E1 23738.989,E2 23738.989} C_VEL
LIN {X 0,Y 503.435,Z 891.609,A -85,B 0,C 180,E1 23736.826,E2 23736.826} C_VEL
LIN {X 0,Y 504.237,Z 858.634,A -85,B 0,C 180,E1 23736.233,E2 23736.233} C_VEL
LIN {X 0,Y 505.327,Z 851.956,A -85,B 0,C 180,E1 23735.635,E2 23735.635} C_VEL
LIN {X 0,Y 509.084,Z 819.748,A -85,B 0,C 180,E1 23732.386,E2 23732.386} C_VEL
LIN {X 0,Y 513.481,Z 793.574,A -85,B 0,C 180,E1 23729.584,E2 23729.584} C_VEL
LIN {X 0,Y 518.497,Z 772.804,A -85,B 0,C 180,E1 23727.189,E2 23727.189} C_VEL
LIN {X 0,Y 524.333,Z 755.979,A -85,B 0,C 180,E1 23725.083,E2 23725.083} C_VEL
LIN {X 0,Y 529.17,Z 745.989,A -85,B 0,C 180,E1 23723.694,E2 23723.694} C_VEL
LIN {X 0,Y 521.376,Z 757.712,A -85,B 0,C 180,E1 23722.423,E2 23722.423} C_VEL
LIN {X 0,Y 516.249,Z 769.075,A -85,B 0,C 180,E1 23721.22,E2 23721.22} C_VEL
LIN {X 0,Y 513.308,Z 780.711,A -85,B 0,C 180,E1 23720.031,E2 23720.031} C_VEL
LIN {X 0,Y 512.459,Z 792.535,A -85,B 0,C 180,E1 23718.862,E2 23718.862} C_VEL
LIN {X 0,Y 513.733,Z 804.741,A -85,B 0,C 180,E1 23717.67,E2 23717.67} C_VEL
LIN {X 0,Y 517.147,Z 816.662,A -85,B 0,C 180,E1 23716.505,E2 23716.505} C_VEL
LIN {X 0,Y 522.035,Z 826.881,A -85,B 0,C 180,E1 23715.493,E2 23715.493} C_VEL
LIN {X 0,Y 528.67,Z 836.443,A -85,B 0,C 180,E1 23714.52,E2 23714.52} C_VEL
LIN {X 0,Y 537.038,Z 845.253,A -85,B 0,C 180,E1 23713.595,E2 23713.595} C_VEL
LIN {X 0,Y 547.203,Z 853.185,A -85,B 0,C 180,E1 23712.732,E2 23712.732} C_VEL
LIN {X 0,Y 558.978,Z 859.818,A -85,B 0,C 180,E1 23711.918,E2 23711.918} C_VEL
LIN {X 0,Y 564.653,Z 862.02,A -85,B 0,C 180,E1 23711.494,E2 23711.494} C_VEL
LIN {X 0,Y 569.316,Z 862.936,A -85,B 0,C 180,E1 23710.959,E2 23710.959} C_VEL
LIN {X 0,Y 572.583,Z 862.637,A -85,B 0,C 180,E1 23710.38,E2 23710.38} C_VEL
LIN {X 0,Y 574.588,Z 861.229,A -85,B 0,C 180,E1 23709.724,E2 23709.724} C_VEL
LIN {X 0,Y 574.945,Z 858.866,A -85,B 0,C 180,E1 23709.08,E2 23709.08} C_VEL
LIN {X 0,Y 574.229,Z 856.913,A -85,B 0,C 180,E1 23708.666,E2 23708.666} C_VEL
LIN {X 0,Y 569.075,Z 877.808,A -85,B 0,C 180,E1 23708.364,E2 23708.364} C_VEL
LIN {X 0,Y 565.539,Z 890.037,A -85,B 0,C 180,E1 23708.073,E2 23708.073} C_VEL
LIN {X 0,Y 559.032,Z 910.121,A -85,B 0,C 180,E1 23708.004,E2 23708.004} C_VEL
LIN {X 0,Y 550.63,Z 930.318,A -85,B 0,C 180,E1 23707.862,E2 23707.862} C_VEL
LIN {X 0,Y 541.57,Z 949.166,A -85,B 0,C 180,E1 23707.591,E2 23707.591} C_VEL
LIN {X 0,Y 534.288,Z 964.788,A -85,B 0,C 180,E1 23707.19,E2 23707.19} C_VEL
LIN {X 0,Y 529.809,Z 976.829,A -85,B 0,C 180,E1 23706.745,E2 23706.745} C_VEL
LIN {X 0,Y 522.608,Z 992.331,A -85,B 0,C 180,E1 23706.241,E2 23706.241} C_VEL
LIN {X 0,Y 518.592,Z 1004.155,A -85,B 0,C 180,E1 23705.746,E2 23705.746} C_VEL
LIN {X 0,Y 514.317,Z 1016.941,A -85,B 0,C 180,E1 23705.199,E2 23705.199} C_VEL
LIN {X 0,Y 512.174,Z 1025.883,A -85,B 0,C 180,E1 23704.802,E2 23704.802} C_VEL
LIN {X 0,Y 511.638,Z 1066.182,A -85,B 0,C 180,E1 23704.175,E2 23704.175} C_VEL
LIN {X 0,Y 510.858,Z 1087.161,A -85,B 0,C 180,E1 23703.658,E2 23703.658} C_VEL
LIN {X 0,Y 509.738,Z 1108.792,A -85,B 0,C 180,E1 23702.91,E2 23702.91} C_VEL
LIN {X 0,Y 508.49,Z 1129.075,A -85,B 0,C 180,E1 23702.001,E2 23702.001} C_VEL
LIN {X 0,Y 506.966,Z 1149.805,A -85,B 0,C 180,E1 23700.85,E2 23700.85} C_VEL
LIN {X 0,Y 505.403,Z 1169.911,A -85,B 0,C 180,E1 23699.487,E2 23699.487} C_VEL
LIN {X 0,Y 503.752,Z 1189.098,A -85,B 0,C 180,E1 23697.932,E2 23697.932} C_VEL
LIN {X 0,Y 502.199,Z 1206.854,A -85,B 0,C 180,E1 23696.232,E2 23696.232} C_VEL
LIN {X 0,Y 500.866,Z 1222.126,A -85,B 0,C 180,E1 23694.534,E2 23694.534} C_VEL
LIN {X 0,Y 499.62,Z 1237.341,A -85,B 0,C 180,E1 23692.597,E2 23692.597} C_VEL
LIN {X 0,Y 498.478,Z 1251.805,A -85,B 0,C 180,E1 23690.427,E2 23690.427} C_VEL
LIN {X 0,Y 497.701,Z 1262.878,A -85,B 0,C 180,E1 23688.507,E2 23688.507} C_VEL
LIN {X 0,Y 497.015,Z 1274.226,A -85,B 0,C 180,E1 23686.239,E2 23686.239} C_VEL
LIN {X 0,Y 496.503,Z 1284.488,A -85,B 0,C 180,E1 23683.747,E2 23683.747} C_VEL
LIN {X 0,Y 496.21,Z 1292.114,A -85,B 0,C 180,E1 23681.507,E2 23681.507} C_VEL
LIN {X 0,Y 496.025,Z 1299.124,A -85,B 0,C 180,E1 23678.93,E2 23678.93} C_VEL
LIN {X 0,Y 495.947,Z 1303.81,A -85,B 0,C 180,E1 23676.599,E2 23676.599} C_VEL
LIN {X 0,Y 495.909,Z 1307.227,A -85,B 0,C 180,E1 23674.163,E2 23674.163} C_VEL
LIN {X 0,Y 495.897,Z 1309.179,A -85,B 0,C 180,E1 23671.502,E2 23671.502} C_VEL
LIN {X 0,Y 495.9,Z 1309.341,A -85,B 0,C 180,E1 23669.192,E2 23669.192} C_VEL
LIN {X 0,Y 495.909,Z 1308.198,A -85,B 0,C 180,E1 23666.88,E2 23666.88} C_VEL
LIN {X 0,Y 495.929,Z 1305.169,A -85,B 0,C 180,E1 23664.215,E2 23664.215} C_VEL
LIN {X 0,Y 495.985,Z 1300.72,A -85,B 0,C 180,E1 23661.811,E2 23661.811} C_VEL
LIN {X 0,Y 496.109,Z 1295.516,A -85,B 0,C 180,E1 23659.667,E2 23659.667} C_VEL
LIN {X 0,Y 496.363,Z 1287.757,A -85,B 0,C 180,E1 23657.148,E2 23657.148} C_VEL
LIN {X 0,Y 496.756,Z 1278.839,A -85,B 0,C 180,E1 23654.832,E2 23654.832} C_VEL
LIN {X 0,Y 497.295,Z 1269.362,A -85,B 0,C 180,E1 23652.751,E2 23652.751} C_VEL
LIN {X 0,Y 498.127,Z 1256.91,A -85,B 0,C 180,E1 23650.415,E2 23650.415} C_VEL
LIN {X 0,Y 499.066,Z 1244.018,A -85,B 0,C 180,E1 23648.369,E2 23648.369} C_VEL
LIN {X 0,Y 500.125,Z 1230.933,A -85,B 0,C 180,E1 23646.557,E2 23646.557} C_VEL
LIN {X 0,Y 501.615,Z 1213.731,A -85,B 0,C 180,E1 23644.498,E2 23644.498} C_VEL
LIN {X 0,Y 503.184,Z 1195.835,A -85,B 0,C 180,E1 23642.677,E2 23642.677} C_VEL
LIN {X 0,Y 504.749,Z 1177.512,A -85,B 0,C 180,E1 23641.097,E2 23641.097} C_VEL
LIN {X 0,Y 506.322,Z 1158.332,A -85,B 0,C 180,E1 23639.699,E2 23639.699} C_VEL
LIN {X 0,Y 507.822,Z 1138.406,A -85,B 0,C 180,E1 23638.488,E2 23638.488} C_VEL
LIN {X 0,Y 509.23,Z 1117.488,A -85,B 0,C 180,E1 23637.454,E2 23637.454} C_VEL
LIN {X 0,Y 510.447,Z 1095.932,A -85,B 0,C 180,E1 23636.618,E2 23636.618} C_VEL
LIN {X 0,Y 511.389,Z 1074.044,A -85,B 0,C 180,E1 23635.991,E2 23635.991} C_VEL
LIN {X 0,Y 511.964,Z 1050.199,A -85,B 0,C 180,E1 23635.552,E2 23635.552} C_VEL
LIN {X 0,Y 512.325,Z 1024.79,A -85,B 0,C 180,E1 23635.158,E2 23635.158} C_VEL
LIN {X 0,Y 516.78,Z 1009.245,A -85,B 0,C 180,E1 23634.452,E2 23634.452} C_VEL
LIN {X 0,Y 519.748,Z 1000.308,A -85,B 0,C 180,E1 23634.075,E2 23634.075} C_VEL
LIN {X 0,Y 524.675,Z 987.553,A -85,B 0,C 180,E1 23633.587,E2 23633.587} C_VEL
LIN {X 0,Y 529.804,Z 976.847,A -85,B 0,C 180,E1 23633.256,E2 23633.256} C_VEL
LIN {X 0,Y 534.28,Z 964.806,A -85,B 0,C 180,E1 23632.81,E2 23632.81} C_VEL
LIN {X 0,Y 541.566,Z 949.175,A -85,B 0,C 180,E1 23632.409,E2 23632.409} C_VEL
LIN {X 0,Y 550.618,Z 930.343,A -85,B 0,C 180,E1 23632.138,E2 23632.138} C_VEL
LIN {X 0,Y 559.02,Z 910.153,A -85,B 0,C 180,E1 23631.996,E2 23631.996} C_VEL
LIN {X 0,Y 565.693,Z 889.475,A -85,B 0,C 180,E1 23631.925,E2 23631.925} C_VEL
LIN {X 0,Y 570.082,Z 874.116,A -85,B 0,C 180,E1 23631.569,E2 23631.569} C_VEL
LIN {X 0,Y 574.299,Z 856.867,A -85,B 0,C 180,E1 23631.317,E2 23631.317} C_VEL
LIN {X 0,Y 575.004,Z 859.806,A -85,B 0,C 180,E1 23630.696,E2 23630.696} C_VEL
LIN {X 0,Y 574.332,Z 861.576,A -85,B 0,C 180,E1 23630.151,E2 23630.151} C_VEL
LIN {X 0,Y 572.475,Z 862.673,A -85,B 0,C 180,E1 23629.596,E2 23629.596} C_VEL
LIN {X 0,Y 569.313,Z 862.945,A -85,B 0,C 180,E1 23629.042,E2 23629.042} C_VEL
LIN {X 0,Y 564.651,Z 862.026,A -85,B 0,C 180,E1 23628.506,E2 23628.506} C_VEL
LIN {X 0,Y 554.668,Z 858.173,A -85,B 0,C 180,E1 23627.499,E2 23627.499} C_VEL
LIN {X 0,Y 545.477,Z 852.63,A -85,B 0,C 180,E1 23626.388,E2 23626.388} C_VEL
LIN {X 0,Y 537.742,Z 845.784,A -85,B 0,C 180,E1 23625.257,E2 23625.257} C_VEL
LIN {X 0,Y 530.948,Z 836.957,A -85,B 0,C 180,E1 23624.018,E2 23624.018} C_VEL
LIN {X 0,Y 525.816,Z 826.715,A -85,B 0,C 180,E1 23622.779,E2 23622.779} C_VEL
LIN {X 0,Y 522.146,Z 814.561,A -85,B 0,C 180,E1 23621.495,E2 23621.495} C_VEL
LIN {X 0,Y 520.086,Z 800.219,A -85,B 0,C 180,E1 23620.165,E2 23620.165} C_VEL
LIN {X 0,Y 519.78,Z 783.857,A -85,B 0,C 180,E1 23618.826,E2 23618.826} C_VEL
LIN {X 0,Y 523.293,Z 734.049,A -85,B 0,C 180,E1 23615.108,E2 23615.108} C_VEL
LIN {X 0,Y 524.042,Z 722.949,A -85,B 0,C 180,E1 23614.253,E2 23614.253} C_VEL
LIN {X 0,Y 514.86,Z 705.892,A -85,B 0,C 180,E1 23611.493,E2 23611.493} C_VEL
LIN {X 0,Y 507.027,Z 691.778,A -85,B 0,C 180,E1 23609.02,E2 23609.02} C_VEL
LIN {X 0,Y 503.987,Z 686.541,A -85,B 0,C 180,E1 23608.046,E2 23608.046} C_VEL
LIN {X 0,Y 501.774,Z 682.378,A -85,B 0,C 180,E1 23607.278,E2 23607.278} C_VEL
LIN {X 0,Y 499.662,Z 678.569,A -85,B 0,C 180,E1 23606.56,E2 23606.56} C_VEL
LIN {X 0,Y 497.089,Z 674.314,A -85,B 0,C 180,E1 23605.696,E2 23605.696} C_VEL
LIN {X 0,Y 496.767,Z 672.855,A -85,B 0,C 180,E1 23605.449,E2 23605.449} C_VEL
LIN {X 0,Y 496.766,Z 672.853,A -85,B 0,C 180,E1 23601.861,E2 23601.861} C_VEL
LIN {X 0,Y 496.761,Z 672.857,A -85,B 0,C 180,E1 23598.3,E2 23598.3} C_VEL
LIN {X 0,Y 496.763,Z 672.859,A -85,B 0,C 180,E1 23594.81,E2 23594.81} C_VEL
LIN {X 0,Y 496.766,Z 672.856,A -85,B 0,C 180,E1 23591.141,E2 23591.141} C_VEL
LIN {X 0,Y 496.756,Z 672.857,A -85,B 0,C 180,E1 23587.634,E2 23587.634} C_VEL
LIN {X 0,Y 496.769,Z 672.856,A -85,B 0,C 180,E1 23584.155,E2 23584.155} C_VEL
LIN {X 0,Y 496.77,Z 672.852,A -85,B 0,C 180,E1 23580.461,E2 23580.461} C_VEL
LIN {X 0,Y 496.758,Z 672.858,A -85,B 0,C 180,E1 23576.884,E2 23576.884} C_VEL
LIN {X 0,Y 496.768,Z 672.856,A -85,B 0,C 180,E1 23573.412,E2 23573.412} C_VEL
LIN {X 0,Y 496.771,Z 672.854,A -85,B 0,C 180,E1 23569.798,E2 23569.798} C_VEL
LIN {X 0,Y 496.758,Z 672.854,A -85,B 0,C 180,E1 23566.26,E2 23566.26} C_VEL
LIN {X 0,Y 496.77,Z 672.859,A -85,B 0,C 180,E1 23562.669,E2 23562.669} C_VEL
LIN {X 0,Y 496.773,Z 672.855,A -85,B 0,C 180,E1 23559.006,E2 23559.006} C_VEL
LIN {X 0,Y 496.758,Z 672.856,A -85,B 0,C 180,E1 23555.377,E2 23555.377} C_VEL
LIN {X 0,Y 496.769,Z 672.826,A -85,B 0,C 180,E1 23551.831,E2 23551.831} C_VEL
LIN {X 0,Y 496.768,Z 672.856,A -85,B 0,C 180,E1 23548.142,E2 23548.142} C_VEL
LIN {X 0,Y 496.753,Z 672.83,A -85,B 0,C 180,E1 23544.571,E2 23544.571} C_VEL
LIN {X 0,Y 496.772,Z 672.853,A -85,B 0,C 180,E1 23541.099,E2 23541.099} C_VEL
LIN {X 0,Y 496.77,Z 672.854,A -85,B 0,C 180,E1 23537.446,E2 23537.446} C_VEL
LIN {X 0,Y 496.758,Z 672.862,A -85,B 0,C 180,E1 23533.819,E2 23533.819} C_VEL
LIN {X 0,Y 496.782,Z 672.965,A -85,B 0,C 180,E1 23531.958,E2 23531.958} C_VEL
LIN {X 0,Y 497.746,Z 675.819,A -85,B 0,C 180,E1 23531.646,E2 23531.646} C_VEL
LIN {X 0,Y 503.74,Z 688.909,A -85,B 0,C 180,E1 23530.078,E2 23530.078} C_VEL
LIN {X 0,Y 508.077,Z 699.007,A -85,B 0,C 180,E1 23528.898,E2 23528.898} C_VEL
LIN {X 0,Y 508.443,Z 702.469,A -85,B 0,C 180,E1 23528.597,E2 23528.597} C_VEL
LIN {X 0,Y 507.07,Z 708.334,A -85,B 0,C 180,E1 23528.263,E2 23528.263} C_VEL
LIN {X 0,Y 504.155,Z 717.245,A -85,B 0,C 180,E1 23527.828,E2 23527.828} C_VEL
LIN {X 0,Y 503.781,Z 719.908,A -85,B 0,C 180,E1 23527.654,E2 23527.654} C_VEL
LIN {X 0,Y 501.986,Z 764.017,A -85,B 0,C 180,E1 23524.517,E2 23524.517} C_VEL
LIN {X 0,Y 502.003,Z 769.529,A -85,B 0,C 180,E1 23524.178,E2 23524.178} C_VEL
LIN {X 0,Y 504.393,Z 785.848,A -85,B 0,C 180,E1 23523.715,E2 23523.715} C_VEL
LIN {X 0,Y 501.034,Z 1020.147,A -85,B 0,C 180,E1 23520.073,E2 23520.073} C_VEL
LIN {X 0,Y 500.489,Z 1041.047,A -85,B 0,C 180,E1 23519.636,E2 23519.636} C_VEL
LIN {X 0,Y 499.649,Z 1061.39,A -85,B 0,C 180,E1 23519,E2 23519} C_VEL
LIN {X 0,Y 498.614,Z 1080.788,A -85,B 0,C 180,E1 23518.179,E2 23518.179} C_VEL
LIN {X 0,Y 497.454,Z 1098.876,A -85,B 0,C 180,E1 23517.21,E2 23517.21} C_VEL
LIN {X 0,Y 496.095,Z 1117.346,A -85,B 0,C 180,E1 23515.986,E2 23515.986} C_VEL
LIN {X 0,Y 494.637,Z 1135.172,A -85,B 0,C 180,E1 23514.545,E2 23514.545} C_VEL
LIN {X 0,Y 493.243,Z 1151.434,A -85,B 0,C 180,E1 23512.967,E2 23512.967} C_VEL
LIN {X 0,Y 491.961,Z 1166.299,A -85,B 0,C 180,E1 23511.26,E2 23511.26} C_VEL
LIN {X 0,Y 490.8,Z 1180.088,A -85,B 0,C 180,E1 23509.393,E2 23509.393} C_VEL
LIN {X 0,Y 489.814,Z 1192.938,A -85,B 0,C 180,E1 23507.339,E2 23507.339} C_VEL
LIN {X 0,Y 489.095,Z 1204.324,A -85,B 0,C 180,E1 23505.222,E2 23505.222} C_VEL
LIN {X 0,Y 488.57,Z 1214.216,A -85,B 0,C 180,E1 23503.009,E2 23503.009} C_VEL
LIN {X 0,Y 488.218,Z 1222.826,A -85,B 0,C 180,E1 23500.621,E2 23500.621} C_VEL
LIN {X 0,Y 488.019,Z 1229.408,A -85,B 0,C 180,E1 23498.279,E2 23498.279} C_VEL
LIN {X 0,Y 487.943,Z 1234.182,A -85,B 0,C 180,E1 23495.998,E2 23495.998} C_VEL
LIN {X 0,Y 487.914,Z 1237.517,A -85,B 0,C 180,E1 23493.634,E2 23493.634} C_VEL
LIN {X 0,Y 487.905,Z 1239.244,A -85,B 0,C 180,E1 23491.291,E2 23491.291} C_VEL
LIN {X 0,Y 487.912,Z 1239.313,A -85,B 0,C 180,E1 23488.943,E2 23488.943} C_VEL
LIN {X 0,Y 487.912,Z 1237.822,A -85,B 0,C 180,E1 23486.592,E2 23486.592} C_VEL
LIN {X 0,Y 487.942,Z 1234.541,A -85,B 0,C 180,E1 23484.119,E2 23484.119} C_VEL
LIN {X 0,Y 488.012,Z 1230.016,A -85,B 0,C 180,E1 23481.872,E2 23481.872} C_VEL
LIN {X 0,Y 488.199,Z 1223.329,A -85,B 0,C 180,E1 23479.442,E2 23479.442} C_VEL
LIN {X 0,Y 488.535,Z 1215.027,A -85,B 0,C 180,E1 23477.109,E2 23477.109} C_VEL
LIN {X 0,Y 489.022,Z 1205.557,A -85,B 0,C 180,E1 23474.949,E2 23474.949} C_VEL
LIN {X 0,Y 489.73,Z 1194.132,A -85,B 0,C 180,E1 23472.78,E2 23472.78} C_VEL
LIN {X 0,Y 490.75,Z 1180.672,A -85,B 0,C 180,E1 23470.603,E2 23470.603} C_VEL
LIN {X 0,Y 491.95,Z 1166.425,A -85,B 0,C 180,E1 23468.665,E2 23468.665} C_VEL
LIN {X 0,Y 493.27,Z 1151.089,A -85,B 0,C 180,E1 23466.907,E2 23466.907} C_VEL
LIN {X 0,Y 494.643,Z 1135.086,A -85,B 0,C 180,E1 23465.357,E2 23465.357} C_VEL
LIN {X 0,Y 496.083,Z 1117.513,A -85,B 0,C 180,E1 23463.935,E2 23463.935} C_VEL
LIN {X 0,Y 497.424,Z 1099.248,A -85,B 0,C 180,E1 23462.722,E2 23462.722} C_VEL
LIN {X 0,Y 498.585,Z 1081.243,A -85,B 0,C 180,E1 23461.753,E2 23461.753} C_VEL
LIN {X 0,Y 499.667,Z 1061.019,A -85,B 0,C 180,E1 23460.897,E2 23460.897} C_VEL
LIN {X 0,Y 500.503,Z 1040.34,A -85,B 0,C 180,E1 23460.256,E2 23460.256} C_VEL
LIN {X 0,Y 501.052,Z 1019.041,A -85,B 0,C 180,E1 23459.82,E2 23459.82} C_VEL
LIN {X 0,Y 504.317,Z 790.898,A -85,B 0,C 180,E1 23456.274,E2 23456.274} C_VEL
LIN {X 0,Y 499.644,Z 770.436,A -85,B 0,C 180,E1 23455.535,E2 23455.535} C_VEL
LIN {X 0,Y 500.864,Z 738.61,A -85,B 0,C 180,E1 23452.348,E2 23452.348} C_VEL
LIN {X 0,Y 502.301,Z 709.661,A -85,B 0,C 180,E1 23449.271,E2 23449.271} C_VEL
LIN {X 0,Y 496.004,Z 692.074,A -85,B 0,C 180,E1 23446.695,E2 23446.695} C_VEL
LIN {X 0,Y 490.329,Z 677.604,A -85,B 0,C 180,E1 23444.545,E2 23444.545} C_VEL
LIN {X 0,Y 488.858,Z 674.032,A -85,B 0,C 180,E1 23444.002,E2 23444.002} C_VEL
LIN {X 0,Y 488.833,Z 673.833,A -85,B 0,C 180,E1 23440.421,E2 23440.421} C_VEL
LIN {X 0,Y 488.837,Z 673.909,A -85,B 0,C 180,E1 23439.884,E2 23439.884} C_VEL
LIN {X 0,Y 490.19,Z 677.403,A -85,B 0,C 180,E1 23439.37,E2 23439.37} C_VEL
LIN {X 0,Y 497.696,Z 695.476,A -85,B 0,C 180,E1 23436.718,E2 23436.718} C_VEL
LIN {X 0,Y 502.746,Z 709.057,A -85,B 0,C 180,E1 23434.875,E2 23434.875} C_VEL
LIN {X 0,Y 500.416,Z 746.254,A -85,B 0,C 180,E1 23431.433,E2 23431.433} C_VEL
LIN {X 0,Y 498.179,Z 784.533,A -85,B 0,C 180,E1 23427.953,E2 23427.953} C_VEL
LIN {X 0,Y 496.022,Z 824.775,A -85,B 0,C 180,E1 23424.339,E2 23424.339} C_VEL
LIN {X 0,Y 494.866,Z 850.429,A -85,B 0,C 180,E1 23422.091,E2 23422.091} C_VEL
LIN {X 0,Y 496.07,Z 860.705,A -85,B 0,C 180,E1 23421.839,E2 23421.839} C_VEL
LIN {X 0,Y 493.924,Z 1019.792,A -85,B 0,C 180,E1 23419.274,E2 23419.274} C_VEL
LIN {X 0,Y 493.501,Z 1038.198,A -85,B 0,C 180,E1 23418.739,E2 23418.739} C_VEL
LIN {X 0,Y 492.974,Z 1053.792,A -85,B 0,C 180,E1 23418.079,E2 23418.079} C_VEL
LIN {X 0,Y 492.342,Z 1068.78,A -85,B 0,C 180,E1 23417.248,E2 23417.248} C_VEL
LIN {X 0,Y 491.545,Z 1084.579,A -85,B 0,C 180,E1 23416.121,E2 23416.121} C_VEL
LIN {X 0,Y 490.819,Z 1097.855,A -85,B 0,C 180,E1 23414.934,E2 23414.934} C_VEL
LIN {X 0,Y 490.08,Z 1110.91,A -85,B 0,C 180,E1 23413.509,E2 23413.509} C_VEL
LIN {X 0,Y 489.4,Z 1122.976,A -85,B 0,C 180,E1 23411.87,E2 23411.87} C_VEL
LIN {X 0,Y 488.91,Z 1132.036,A -85,B 0,C 180,E1 23410.363,E2 23410.363} C_VEL
LIN {X 0,Y 488.508,Z 1140.744,A -85,B 0,C 180,E1 23408.593,E2 23408.593} C_VEL
LIN {X 0,Y 488.224,Z 1148.296,A -85,B 0,C 180,E1 23406.586,E2 23406.586} C_VEL
LIN {X 0,Y 488.084,Z 1153.283,A -85,B 0,C 180,E1 23404.818,E2 23404.818} C_VEL
LIN {X 0,Y 488,Z 1157.144,A -85,B 0,C 180,E1 23402.936,E2 23402.936} C_VEL
LIN {X 0,Y 487.968,Z 1159.615,A -85,B 0,C 180,E1 23400.822,E2 23400.822} C_VEL
LIN {X 0,Y 487.967,Z 1160.31,A -85,B 0,C 180,E1 23398.944,E2 23398.944} C_VEL
LIN {X 0,Y 487.977,Z 1159.665,A -85,B 0,C 180,E1 23397.064,E2 23397.064} C_VEL
LIN {X 0,Y 488.031,Z 1157.057,A -85,B 0,C 180,E1 23394.828,E2 23394.828} C_VEL
LIN {X 0,Y 488.146,Z 1153.189,A -85,B 0,C 180,E1 23392.941,E2 23392.941} C_VEL
LIN {X 0,Y 488.299,Z 1148.161,A -85,B 0,C 180,E1 23391.166,E2 23391.166} C_VEL
LIN {X 0,Y 488.633,Z 1140.548,A -85,B 0,C 180,E1 23389.149,E2 23389.149} C_VEL
LIN {X 0,Y 489.065,Z 1132.446,A -85,B 0,C 180,E1 23387.484,E2 23387.484} C_VEL
LIN {X 0,Y 489.663,Z 1122.464,A -85,B 0,C 180,E1 23385.817,E2 23385.817} C_VEL
LIN {X 0,Y 490.379,Z 1110.755,A -85,B 0,C 180,E1 23384.236,E2 23384.236} C_VEL
LIN {X 0,Y 491.157,Z 1097.863,A -85,B 0,C 180,E1 23382.832,E2 23382.832} C_VEL
LIN {X 0,Y 491.942,Z 1083.479,A -85,B 0,C 180,E1 23381.576,E2 23381.576} C_VEL
LIN {X 0,Y 492.648,Z 1068.816,A -85,B 0,C 180,E1 23380.559,E2 23380.559} C_VEL
LIN {X 0,Y 493.261,Z 1053.265,A -85,B 0,C 180,E1 23379.719,E2 23379.719} C_VEL
LIN {X 0,Y 493.713,Z 1036.764,A -85,B 0,C 180,E1 23379.069,E2 23379.069} C_VEL
LIN {X 0,Y 493.962,Z 1019.657,A -85,B 0,C 180,E1 23378.625,E2 23378.625} C_VEL
LIN {X 0,Y 495.89,Z 911.712,A -85,B 0,C 180,E1 23376.756,E2 23376.756} C_VEL
LIN {X 0,Y 497.312,Z 862.189,A -85,B 0,C 180,E1 23375.818,E2 23375.818} C_VEL
LIN {X 0,Y 498.704,Z 857.111,A -85,B 0,C 180,E1 23375.417,E2 23375.417} C_VEL
LIN {X 0,Y 502.97,Z 824.077,A -85,B 0,C 180,E1 23372.021,E2 23372.021} C_VEL
LIN {X 0,Y 507.761,Z 798.395,A -85,B 0,C 180,E1 23369.205,E2 23369.205} C_VEL
LIN {X 0,Y 513.182,Z 778.133,A -85,B 0,C 180,E1 23366.806,E2 23366.806} C_VEL
LIN {X 0,Y 519.027,Z 762.798,A -85,B 0,C 180,E1 23364.831,E2 23364.831} C_VEL
LIN {X 0,Y 522.795,Z 755.419,A -85,B 0,C 180,E1 23363.813,E2 23363.813} C_VEL
LIN {X 0,Y 515.201,Z 766.783,A -85,B 0,C 180,E1 23362.538,E2 23362.538} C_VEL
LIN {X 0,Y 510.066,Z 778.124,A -85,B 0,C 180,E1 23361.278,E2 23361.278} C_VEL
LIN {X 0,Y 507.316,Z 789.372,A -85,B 0,C 180,E1 23360.056,E2 23360.056} C_VEL
LIN {X 0,Y 506.727,Z 800.776,A -85,B 0,C 180,E1 23358.849,E2 23358.849} C_VEL
LIN {X 0,Y 508.244,Z 812.38,A -85,B 0,C 180,E1 23357.64,E2 23357.64} C_VEL
LIN {X 0,Y 512.006,Z 824.113,A -85,B 0,C 180,E1 23356.422,E2 23356.422} C_VEL
LIN {X 0,Y 517.665,Z 834.838,A -85,B 0,C 180,E1 23355.299,E2 23355.299} C_VEL
LIN {X 0,Y 525.673,Z 845.225,A -85,B 0,C 180,E1 23354.187,E2 23354.187} C_VEL
LIN {X 0,Y 534.297,Z 853.425,A -85,B 0,C 180,E1 23353.285,E2 23353.285} C_VEL
LIN {X 0,Y 544.643,Z 860.906,A -85,B 0,C 180,E1 23352.44,E2 23352.44} C_VEL
LIN {X 0,Y 556.537,Z 867.214,A -85,B 0,C 180,E1 23351.637,E2 23351.637} C_VEL
LIN {X 0,Y 562.248,Z 869.318,A -85,B 0,C 180,E1 23351.216,E2 23351.216} C_VEL
LIN {X 0,Y 566.96,Z 870.164,A -85,B 0,C 180,E1 23350.684,E2 23350.684} C_VEL
LIN {X 0,Y 570.161,Z 869.853,A -85,B 0,C 180,E1 23350.13,E2 23350.13} C_VEL
LIN {X 0,Y 572.22,Z 868.528,A -85,B 0,C 180,E1 23349.497,E2 23349.497} C_VEL
LIN {X 0,Y 572.47,Z 868.134,A -85,B 0,C 180,E1 23349.33,E2 23349.33} C_VEL
LIN {X 0,Y 566.821,Z 884.888,A -85,B 0,C 180,E1 23349.031,E2 23349.031} C_VEL
LIN {X 0,Y 564.692,Z 891.1,A -85,B 0,C 180,E1 23348.88,E2 23348.88} C_VEL
LIN {X 0,Y 556.073,Z 910.711,A -85,B 0,C 180,E1 23348.776,E2 23348.776} C_VEL
LIN {X 0,Y 545.624,Z 930.572,A -85,B 0,C 180,E1 23348.54,E2 23348.54} C_VEL
LIN {X 0,Y 535.151,Z 949.029,A -85,B 0,C 180,E1 23348.133,E2 23348.133} C_VEL
LIN {X 0,Y 527.322,Z 964.319,A -85,B 0,C 180,E1 23347.629,E2 23347.629} C_VEL
LIN {X 0,Y 522.033,Z 977.42,A -85,B 0,C 180,E1 23347.109,E2 23347.109} C_VEL
LIN {X 0,Y 515.538,Z 990.669,A -85,B 0,C 180,E1 23346.611,E2 23346.611} C_VEL
LIN {X 0,Y 511.187,Z 1003.26,A -85,B 0,C 180,E1 23346.068,E2 23346.068} C_VEL
LIN {X 0,Y 506.888,Z 1016.002,A -85,B 0,C 180,E1 23345.515,E2 23345.515} C_VEL
LIN {X 0,Y 504.891,Z 1024.044,A -85,B 0,C 180,E1 23345.172,E2 23345.172} C_VEL
LIN {X 0,Y 504.281,Z 1066.405,A -85,B 0,C 180,E1 23344.529,E2 23344.529} C_VEL
LIN {X 0,Y 503.452,Z 1090.896,A -85,B 0,C 180,E1 23343.942,E2 23343.942} C_VEL
LIN {X 0,Y 502.576,Z 1111.933,A -85,B 0,C 180,E1 23343.237,E2 23343.237} C_VEL
LIN {X 0,Y 501.528,Z 1130.142,A -85,B 0,C 180,E1 23342.432,E2 23342.432} C_VEL
LIN {X 0,Y 499.994,Z 1149.804,A -85,B 0,C 180,E1 23341.328,E2 23341.328} C_VEL
LIN {X 0,Y 498.328,Z 1169.603,A -85,B 0,C 180,E1 23339.974,E2 23339.974} C_VEL
LIN {X 0,Y 496.595,Z 1188.218,A -85,B 0,C 180,E1 23338.456,E2 23338.456} C_VEL
LIN {X 0,Y 494.931,Z 1205.872,A -85,B 0,C 180,E1 23336.757,E2 23336.757} C_VEL
LIN {X 0,Y 493.463,Z 1221.098,A -85,B 0,C 180,E1 23335.055,E2 23335.055} C_VEL
LIN {X 0,Y 492.237,Z 1234.588,A -85,B 0,C 180,E1 23333.335,E2 23333.335} C_VEL
LIN {X 0,Y 490.953,Z 1249.607,A -85,B 0,C 180,E1 23331.13,E2 23331.13} C_VEL
LIN {X 0,Y 489.941,Z 1262.226,A -85,B 0,C 180,E1 23328.935,E2 23328.935} C_VEL
LIN {X 0,Y 489.236,Z 1272.505,A -85,B 0,C 180,E1 23326.871,E2 23326.871} C_VEL
LIN {X 0,Y 488.635,Z 1283.179,A -85,B 0,C 180,E1 23324.336,E2 23324.336} C_VEL
LIN {X 0,Y 488.27,Z 1291.368,A -85,B 0,C 180,E1 23321.937,E2 23321.937} C_VEL
LIN {X 0,Y 488.072,Z 1297.674,A -85,B 0,C 180,E1 23319.671,E2 23319.671} C_VEL
LIN {X 0,Y 487.957,Z 1303.42,A -85,B 0,C 180,E1 23316.944,E2 23316.944} C_VEL
LIN {X 0,Y 487.918,Z 1306.813,A -85,B 0,C 180,E1 23314.584,E2 23314.584} C_VEL
LIN {X 0,Y 487.908,Z 1308.91,A -85,B 0,C 180,E1 23312.114,E2 23312.114} C_VEL
LIN {X 0,Y 487.895,Z 1309.393,A -85,B 0,C 180,E1 23309.413,E2 23309.413} C_VEL
LIN {X 0,Y 487.901,Z 1308.442,A -85,B 0,C 180,E1 23307.181,E2 23307.181} C_VEL
LIN {X 0,Y 487.923,Z 1305.979,A -85,B 0,C 180,E1 23304.71,E2 23304.71} C_VEL
LIN {X 0,Y 487.991,Z 1301.644,A -85,B 0,C 180,E1 23302.11,E2 23302.11} C_VEL
LIN {X 0,Y 488.108,Z 1296.448,A -85,B 0,C 180,E1 23299.854,E2 23299.854} C_VEL
LIN {X 0,Y 488.351,Z 1289.507,A -85,B 0,C 180,E1 23297.466,E2 23297.466} C_VEL
LIN {X 0,Y 488.804,Z 1279.845,A -85,B 0,C 180,E1 23294.822,E2 23294.822} C_VEL
LIN {X 0,Y 489.391,Z 1270.213,A -85,B 0,C 180,E1 23292.646,E2 23292.646} C_VEL
LIN {X 0,Y 490.263,Z 1258.32,A -85,B 0,C 180,E1 23290.336,E2 23290.336} C_VEL
LIN {X 0,Y 491.348,Z 1244.676,A -85,B 0,C 180,E1 23288.113,E2 23288.113} C_VEL
LIN {X 0,Y 492.473,Z 1231.846,A -85,B 0,C 180,E1 23286.298,E2 23286.298} C_VEL
LIN {X 0,Y 493.988,Z 1215.963,A -85,B 0,C 180,E1 23284.333,E2 23284.333} C_VEL
LIN {X 0,Y 495.704,Z 1197.731,A -85,B 0,C 180,E1 23282.426,E2 23282.426} C_VEL
LIN {X 0,Y 497.457,Z 1179.054,A -85,B 0,C 180,E1 23280.764,E2 23280.764} C_VEL
LIN {X 0,Y 499.22,Z 1159.252,A -85,B 0,C 180,E1 23279.289,E2 23279.289} C_VEL
LIN {X 0,Y 500.865,Z 1139.056,A -85,B 0,C 180,E1 23278.039,E2 23278.039} C_VEL
LIN {X 0,Y 502.12,Z 1120.276,A -85,B 0,C 180,E1 23277.107,E2 23277.107} C_VEL
LIN {X 0,Y 503.381,Z 1097.211,A -85,B 0,C 180,E1 23276.214,E2 23276.214} C_VEL
LIN {X 0,Y 504.377,Z 1074.305,A -85,B 0,C 180,E1 23275.556,E2 23275.556} C_VEL
LIN {X 0,Y 505.043,Z 1050.629,A -85,B 0,C 180,E1 23275.103,E2 23275.103} C_VEL
LIN {X 0,Y 505.496,Z 1023.943,A -85,B 0,C 180,E1 23274.686,E2 23274.686} C_VEL
LIN {X 0,Y 510.031,Z 1008.596,A -85,B 0,C 180,E1 23273.977,E2 23273.977} C_VEL
LIN {X 0,Y 516.286,Z 990.783,A -85,B 0,C 180,E1 23273.244,E2 23273.244} C_VEL
LIN {X 0,Y 523.448,Z 975.35,A -85,B 0,C 180,E1 23272.735,E2 23272.735} C_VEL
LIN {X 0,Y 528.289,Z 962.926,A -85,B 0,C 180,E1 23272.271,E2 23272.271} C_VEL
LIN {X 0,Y 536.673,Z 946.329,A -85,B 0,C 180,E1 23271.791,E2 23271.791} C_VEL
LIN {X 0,Y 547.504,Z 927.2,A -85,B 0,C 180,E1 23271.409,E2 23271.409} C_VEL
LIN {X 0,Y 557.731,Z 907.24,A -85,B 0,C 180,E1 23271.198,E2 23271.198} C_VEL
LIN {X 0,Y 565.292,Z 889.473,A -85,B 0,C 180,E1 23271.1,E2 23271.1} C_VEL
LIN {X 0,Y 569.766,Z 876.245,A -85,B 0,C 180,E1 23270.789,E2 23270.789} C_VEL
LIN {X 0,Y 572.484,Z 868.076,A -85,B 0,C 180,E1 23270.656,E2 23270.656} C_VEL
LIN {X 0,Y 571.017,Z 869.52,A -85,B 0,C 180,E1 23270.08,E2 23270.08} C_VEL
LIN {X 0,Y 568.119,Z 870.175,A -85,B 0,C 180,E1 23269.49,E2 23269.49} C_VEL
LIN {X 0,Y 564.389,Z 869.836,A -85,B 0,C 180,E1 23268.998,E2 23268.998} C_VEL
LIN {X 0,Y 553.495,Z 866.27,A -85,B 0,C 180,E1 23267.94,E2 23267.94} C_VEL
LIN {X 0,Y 543.368,Z 860.898,A -85,B 0,C 180,E1 23266.776,E2 23266.776} C_VEL
LIN {X 0,Y 534.18,Z 853.552,A -85,B 0,C 180,E1 23265.491,E2 23265.491} C_VEL
LIN {X 0,Y 527.142,Z 845.266,A -85,B 0,C 180,E1 23264.267,E2 23264.267} C_VEL
LIN {X 0,Y 521.587,Z 835.681,A -85,B 0,C 180,E1 23263.034,E2 23263.034} C_VEL
LIN {X 0,Y 517.396,Z 824.421,A -85,B 0,C 180,E1 23261.761,E2 23261.761} C_VEL
LIN {X 0,Y 514.679,Z 811.323,A -85,B 0,C 180,E1 23260.455,E2 23260.455} C_VEL
LIN {X 0,Y 513.547,Z 796.128,A -85,B 0,C 180,E1 23259.11,E2 23259.11} C_VEL
LIN {X 0,Y 514.16,Z 777.203,A -85,B 0,C 180,E1 23257.634,E2 23257.634} C_VEL
LIN {X 0,Y 517.388,Z 736.699,A -85,B 0,C 180,E1 23254.59,E2 23254.59} C_VEL
LIN {X 0,Y 517.98,Z 727.264,A -85,B 0,C 180,E1 23253.841,E2 23253.841} C_VEL
LIN {X 0,Y 507.671,Z 707.969,A -85,B 0,C 180,E1 23250.67,E2 23250.67} C_VEL
LIN {X 0,Y 499.229,Z 692.943,A -85,B 0,C 180,E1 23247.947,E2 23247.947} C_VEL
LIN {X 0,Y 496.251,Z 687.779,A -85,B 0,C 180,E1 23246.958,E2 23246.958} C_VEL
LIN {X 0,Y 493.694,Z 683.197,A -85,B 0,C 180,E1 23246.07,E2 23246.07} C_VEL
LIN {X 0,Y 491.824,Z 679.771,A -85,B 0,C 180,E1 23245.401,E2 23245.401} C_VEL
LIN {X 0,Y 490.816,Z 678.21,A -85,B 0,C 180,E1 23245.07,E2 23245.07} C_VEL
LIN {X 0,Y 489.222,Z 675.543,A -85,B 0,C 180,E1 23244.512,E2 23244.512} C_VEL
LIN {X 0,Y 488.827,Z 673.846,A -85,B 0,C 180,E1 23244.211,E2 23244.211} C_VEL
LIN {X 0,Y 488.819,Z 673.844,A -85,B 0,C 180,E1 23240.724,E2 23240.724} C_VEL
LIN {X 0,Y 488.817,Z 673.844,A -85,B 0,C 180,E1 23237.13,E2 23237.13} C_VEL
LIN {X 0,Y 488.827,Z 673.845,A -85,B 0,C 180,E1 23233.605,E2 23233.605} C_VEL
LIN {X 0,Y 488.822,Z 673.845,A -85,B 0,C 180,E1 23230.012,E2 23230.012} C_VEL
LIN {X 0,Y 488.815,Z 673.843,A -85,B 0,C 180,E1 23226.459,E2 23226.459} C_VEL
LIN {X 0,Y 488.821,Z 673.847,A -85,B 0,C 180,E1 23222.931,E2 23222.931} C_VEL
LIN {X 0,Y 488.831,Z 673.847,A -85,B 0,C 180,E1 23219.414,E2 23219.414} C_VEL
LIN {X 0,Y 488.815,Z 673.844,A -85,B 0,C 180,E1 23215.777,E2 23215.777} C_VEL
LIN {X 0,Y 488.818,Z 673.848,A -85,B 0,C 180,E1 23212.241,E2 23212.241} C_VEL
LIN {X 0,Y 488.828,Z 673.846,A -85,B 0,C 180,E1 23208.676,E2 23208.676} C_VEL
LIN {X 0,Y 488.817,Z 673.845,A -85,B 0,C 180,E1 23205.064,E2 23205.064} C_VEL
LIN {X 0,Y 488.818,Z 673.843,A -85,B 0,C 180,E1 23201.515,E2 23201.515} C_VEL
LIN {X 0,Y 488.834,Z 673.842,A -85,B 0,C 180,E1 23197.892,E2 23197.892} C_VEL
LIN {X 0,Y 488.818,Z 673.845,A -85,B 0,C 180,E1 23194.301,E2 23194.301} C_VEL
LIN {X 0,Y 488.813,Z 673.81,A -85,B 0,C 180,E1 23190.857,E2 23190.857} C_VEL
LIN {X 0,Y 488.831,Z 673.846,A -85,B 0,C 180,E1 23187.317,E2 23187.317} C_VEL
LIN {X 0,Y 488.821,Z 673.823,A -85,B 0,C 180,E1 23183.697,E2 23183.697} C_VEL
LIN {X 0,Y 488.814,Z 673.831,A -85,B 0,C 180,E1 23180.19,E2 23180.19} C_VEL
LIN {X 0,Y 488.826,Z 673.848,A -85,B 0,C 180,E1 23176.586,E2 23176.586} C_VEL
LIN {X 0,Y 488.831,Z 673.853,A -85,B 0,C 180,E1 23173.091,E2 23173.091} C_VEL
LIN {X 0,Y 488.841,Z 674.023,A -85,B 0,C 180,E1 23172.661,E2 23172.661} C_VEL
LIN {X 0,Y 490.28,Z 677.552,A -85,B 0,C 180,E1 23172.244,E2 23172.244} C_VEL
LIN {X 0,Y 497.922,Z 694.583,A -85,B 0,C 180,E1 23170.167,E2 23170.167} C_VEL
LIN {X 0,Y 504.241,Z 709.803,A -85,B 0,C 180,E1 23168.4,E2 23168.4} C_VEL
LIN {X 0,Y 503.781,Z 719.908,A -85,B 0,C 180,E1 23167.654,E2 23167.654} C_VEL
LIN {X 0,Y 502.64,Z 726.648,A -85,B 0,C 180,E1 23167.235,E2 23167.235} C_VEL
LIN {X 0,Y 496.589,Z 745.453,A -85,B 0,C 180,E1 23166.331,E2 23166.331} C_VEL
LIN {X 0,Y 495.702,Z 751.264,A -85,B 0,C 180,E1 23165.967,E2 23165.967} C_VEL
LIN {X 0,Y 495.251,Z 769.968,A -85,B 0,C 180,E1 23164.711,E2 23164.711} C_VEL
LIN {X 0,Y 497.757,Z 787.071,A -85,B 0,C 180,E1 23164.213,E2 23164.213} C_VEL
LIN {X 0,Y 494.131,Z 1020.784,A -85,B 0,C 180,E1 23160.533,E2 23160.533} C_VEL
LIN {X 0,Y 493.559,Z 1041.658,A -85,B 0,C 180,E1 23160.091,E2 23160.091} C_VEL
LIN {X 0,Y 492.672,Z 1062.039,A -85,B 0,C 180,E1 23159.446,E2 23159.446} C_VEL
LIN {X 0,Y 491.576,Z 1081.35,A -85,B 0,C 180,E1 23158.62,E2 23158.62} C_VEL
LIN {X 0,Y 490.345,Z 1099.453,A -85,B 0,C 180,E1 23157.638,E2 23157.638} C_VEL
LIN {X 0,Y 488.875,Z 1118.096,A -85,B 0,C 180,E1 23156.387,E2 23156.387} C_VEL
LIN {X 0,Y 487.313,Z 1135.969,A -85,B 0,C 180,E1 23154.921,E2 23154.921} C_VEL
LIN {X 0,Y 485.835,Z 1151.98,A -85,B 0,C 180,E1 23153.345,E2 23153.345} C_VEL
LIN {X 0,Y 484.444,Z 1166.826,A -85,B 0,C 180,E1 23151.617,E2 23151.617} C_VEL
LIN {X 0,Y 483.158,Z 1180.916,A -85,B 0,C 180,E1 23149.679,E2 23149.679} C_VEL
LIN {X 0,Y 482.088,Z 1193.504,A -85,B 0,C 180,E1 23147.626,E2 23147.626} C_VEL
LIN {X 0,Y 481.27,Z 1204.256,A -85,B 0,C 180,E1 23145.545,E2 23145.545} C_VEL
LIN {X 0,Y 480.617,Z 1214.693,A -85,B 0,C 180,E1 23143.106,E2 23143.106} C_VEL
LIN {X 0,Y 480.239,Z 1223.25,A -85,B 0,C 180,E1 23140.67,E2 23140.67} C_VEL
LIN {X 0,Y 480.024,Z 1229.795,A -85,B 0,C 180,E1 23138.263,E2 23138.263} C_VEL
LIN {X 0,Y 479.945,Z 1234.387,A -85,B 0,C 180,E1 23135.978,E2 23135.978} C_VEL
LIN {X 0,Y 479.913,Z 1237.735,A -85,B 0,C 180,E1 23133.463,E2 23133.463} C_VEL
LIN {X 0,Y 479.912,Z 1239.296,A -85,B 0,C 180,E1 23131.074,E2 23131.074} C_VEL
LIN {X 0,Y 479.905,Z 1239.268,A -85,B 0,C 180,E1 23128.686,E2 23128.686} C_VEL
LIN {X 0,Y 479.913,Z 1237.595,A -85,B 0,C 180,E1 23126.296,E2 23126.296} C_VEL
LIN {X 0,Y 479.947,Z 1234.335,A -85,B 0,C 180,E1 23123.9,E2 23123.9} C_VEL
LIN {X 0,Y 480.035,Z 1229.412,A -85,B 0,C 180,E1 23121.495,E2 23121.495} C_VEL
LIN {X 0,Y 480.243,Z 1223.117,A -85,B 0,C 180,E1 23119.2,E2 23119.2} C_VEL
LIN {X 0,Y 480.623,Z 1214.567,A -85,B 0,C 180,E1 23116.771,E2 23116.771} C_VEL
LIN {X 0,Y 481.325,Z 1203.514,A -85,B 0,C 180,E1 23114.209,E2 23114.209} C_VEL
LIN {X 0,Y 482.227,Z 1191.961,A -85,B 0,C 180,E1 23112.004,E2 23112.004} C_VEL
LIN {X 0,Y 483.358,Z 1178.77,A -85,B 0,C 180,E1 23109.907,E2 23109.907} C_VEL
LIN {X 0,Y 484.65,Z 1164.578,A -85,B 0,C 180,E1 23108.01,E2 23108.01} C_VEL
LIN {X 0,Y 486.024,Z 1149.916,A -85,B 0,C 180,E1 23106.349,E2 23106.349} C_VEL
LIN {X 0,Y 487.557,Z 1133.105,A -85,B 0,C 180,E1 23104.741,E2 23104.741} C_VEL
LIN {X 0,Y 488.999,Z 1116.35,A -85,B 0,C 180,E1 23103.398,E2 23103.398} C_VEL
LIN {X 0,Y 490.472,Z 1097.79,A -85,B 0,C 180,E1 23102.171,E2 23102.171} C_VEL
LIN {X 0,Y 491.767,Z 1078.516,A -85,B 0,C 180,E1 23101.15,E2 23101.15} C_VEL
LIN {X 0,Y 492.845,Z 1058.819,A -85,B 0,C 180,E1 23100.346,E2 23100.346} C_VEL
LIN {X 0,Y 493.643,Z 1038.633,A -85,B 0,C 180,E1 23099.741,E2 23099.741} C_VEL
LIN {X 0,Y 494.217,Z 1015.035,A -85,B 0,C 180,E1 23099.287,E2 23099.287} C_VEL
LIN {X 0,Y 497.649,Z 792.403,A -85,B 0,C 180,E1 23095.78,E2 23095.78} C_VEL
LIN {X 0,Y 492.747,Z 771.189,A -85,B 0,C 180,E1 23095.009,E2 23095.009} C_VEL
LIN {X 0,Y 493.91,Z 741.357,A -85,B 0,C 180,E1 23092.018,E2 23092.018} C_VEL
LIN {X 0,Y 495.423,Z 713.177,A -85,B 0,C 180,E1 23089.008,E2 23089.008} C_VEL
LIN {X 0,Y 488.849,Z 694.74,A -85,B 0,C 180,E1 23086.265,E2 23086.265} C_VEL
LIN {X 0,Y 482.451,Z 678.66,A -85,B 0,C 180,E1 23083.805,E2 23083.805} C_VEL
LIN {X 0,Y 481.008,Z 675.569,A -85,B 0,C 180,E1 23083.312,E2 23083.312} C_VEL
LIN {X 0,Y 480.877,Z 674.825,A -85,B 0,C 180,E1 23083.163,E2 23083.163} C_VEL
LIN {X 0,Y 480.888,Z 674.87,A -85,B 0,C 180,E1 23080.663,E2 23080.663} C_VEL
LIN {X 0,Y 482.352,Z 678.524,A -85,B 0,C 180,E1 23080.102,E2 23080.102} C_VEL
LIN {X 0,Y 490.343,Z 697.689,A -85,B 0,C 180,E1 23077.234,E2 23077.234} C_VEL
LIN {X 0,Y 495.887,Z 712.435,A -85,B 0,C 180,E1 23075.181,E2 23075.181} C_VEL
LIN {X 0,Y 493.44,Z 749.607,A -85,B 0,C 180,E1 23071.717,E2 23071.717} C_VEL
LIN {X 0,Y 491.044,Z 788.024,A -85,B 0,C 180,E1 23068.19,E2 23068.19} C_VEL
LIN {X 0,Y 488.768,Z 828.408,A -85,B 0,C 180,E1 23064.537,E2 23064.537} C_VEL
LIN {X 0,Y 487.699,Z 851.598,A -85,B 0,C 180,E1 23062.494,E2 23062.494} C_VEL
LIN {X 0,Y 488.893,Z 861.727,A -85,B 0,C 180,E1 23062.24,E2 23062.24} C_VEL
LIN {X 0,Y 486.438,Z 1021.465,A -85,B 0,C 180,E1 23059.579,E2 23059.579} C_VEL
LIN {X 0,Y 486.006,Z 1039.507,A -85,B 0,C 180,E1 23059.039,E2 23059.039} C_VEL
LIN {X 0,Y 485.431,Z 1055.741,A -85,B 0,C 180,E1 23058.335,E2 23058.335} C_VEL
LIN {X 0,Y 484.701,Z 1071.878,A -85,B 0,C 180,E1 23057.404,E2 23057.404} C_VEL
LIN {X 0,Y 483.861,Z 1087.196,A -85,B 0,C 180,E1 23056.26,E2 23056.26} C_VEL
LIN {X 0,Y 483.071,Z 1100.834,A -85,B 0,C 180,E1 23054.995,E2 23054.995} C_VEL
LIN {X 0,Y 482.285,Z 1113.857,A -85,B 0,C 180,E1 23053.512,E2 23053.512} C_VEL
LIN {X 0,Y 481.628,Z 1124.72,A -85,B 0,C 180,E1 23051.982,E2 23051.982} C_VEL
LIN {X 0,Y 481.066,Z 1134.552,A -85,B 0,C 180,E1 23050.297,E2 23050.297} C_VEL
LIN {X 0,Y 480.597,Z 1143.978,A -85,B 0,C 180,E1 23048.254,E2 23048.254} C_VEL
LIN {X 0,Y 480.342,Z 1150.706,A -85,B 0,C 180,E1 23046.334,E2 23046.334} C_VEL
LIN {X 0,Y 480.175,Z 1156.027,A -85,B 0,C 180,E1 23044.299,E2 23044.299} C_VEL
LIN {X 0,Y 480.106,Z 1159.659,A -85,B 0,C 180,E1 23042.149,E2 23042.149} C_VEL
LIN {X 0,Y 480.084,Z 1161.339,A -85,B 0,C 180,E1 23040.239,E2 23040.239} C_VEL
LIN {X 0,Y 480.086,Z 1161.685,A -85,B 0,C 180,E1 23038.21,E2 23038.21} C_VEL
LIN {X 0,Y 480.131,Z 1160.207,A -85,B 0,C 180,E1 23036.06,E2 23036.06} C_VEL
LIN {X 0,Y 480.215,Z 1157.436,A -85,B 0,C 180,E1 23034.145,E2 23034.145} C_VEL
LIN {X 0,Y 480.397,Z 1152.511,A -85,B 0,C 180,E1 23031.984,E2 23031.984} C_VEL
LIN {X 0,Y 480.674,Z 1146.299,A -85,B 0,C 180,E1 23030.058,E2 23030.058} C_VEL
LIN {X 0,Y 481.089,Z 1138.571,A -85,B 0,C 180,E1 23028.208,E2 23028.208} C_VEL
LIN {X 0,Y 481.732,Z 1128.447,A -85,B 0,C 180,E1 23026.314,E2 23026.314} C_VEL
LIN {X 0,Y 482.417,Z 1117.994,A -85,B 0,C 180,E1 23024.739,E2 23024.739} C_VEL
LIN {X 0,Y 483.216,Z 1105.621,A -85,B 0,C 180,E1 23023.223,E2 23023.223} C_VEL
LIN {X 0,Y 484.046,Z 1092.033,A -85,B 0,C 180,E1 23021.888,E2 23021.888} C_VEL
LIN {X 0,Y 484.853,Z 1077.386,A -85,B 0,C 180,E1 23020.735,E2 23020.735} C_VEL
LIN {X 0,Y 485.502,Z 1062.712,A -85,B 0,C 180,E1 23019.821,E2 23019.821} C_VEL
LIN {X 0,Y 486.057,Z 1046.354,A -85,B 0,C 180,E1 23019.054,E2 23019.054} C_VEL
LIN {X 0,Y 486.402,Z 1029.386,A -85,B 0,C 180,E1 23018.5,E2 23018.5} C_VEL
LIN {X 0,Y 486.693,Z 1005.471,A -85,B 0,C 180,E1 23018.034,E2 23018.034} C_VEL
LIN {X 0,Y 488.725,Z 915.893,A -85,B 0,C 180,E1 23016.392,E2 23016.392} C_VEL
LIN {X 0,Y 490.542,Z 865.566,A -85,B 0,C 180,E1 23015.366,E2 23015.366} C_VEL
LIN {X 0,Y 492.368,Z 860.008,A -85,B 0,C 180,E1 23014.951,E2 23014.951} C_VEL
LIN {X 0,Y 497.017,Z 827.99,A -85,B 0,C 180,E1 23011.591,E2 23011.591} C_VEL
LIN {X 0,Y 502.129,Z 803.359,A -85,B 0,C 180,E1 23008.821,E2 23008.821} C_VEL
LIN {X 0,Y 507.151,Z 785.949,A -85,B 0,C 180,E1 23006.713,E2 23006.713} C_VEL
LIN {X 0,Y 513.12,Z 771.098,A -85,B 0,C 180,E1 23004.776,E2 23004.776} C_VEL
LIN {X 0,Y 516.313,Z 764.985,A -85,B 0,C 180,E1 23003.908,E2 23003.908} C_VEL
LIN {X 0,Y 508.977,Z 775.94,A -85,B 0,C 180,E1 23002.626,E2 23002.626} C_VEL
LIN {X 0,Y 504.172,Z 786.518,A -85,B 0,C 180,E1 23001.386,E2 23001.386} C_VEL
LIN {X 0,Y 501.532,Z 797.381,A -85,B 0,C 180,E1 23000.134,E2 23000.134} C_VEL
LIN {X 0,Y 501.085,Z 808.331,A -85,B 0,C 180,E1 22998.892,E2 22998.892} C_VEL
LIN {X 0,Y 502.691,Z 819.193,A -85,B 0,C 180,E1 22997.687,E2 22997.687} C_VEL
LIN {X 0,Y 506.483,Z 830.435,A -85,B 0,C 180,E1 22996.452,E2 22996.452} C_VEL
LIN {X 0,Y 512.573,Z 841.459,A -85,B 0,C 180,E1 22995.236,E2 22995.236} C_VEL
LIN {X 0,Y 520.728,Z 851.663,A -85,B 0,C 180,E1 22994.101,E2 22994.101} C_VEL
LIN {X 0,Y 530.097,Z 860.282,A -85,B 0,C 180,E1 22993.118,E2 22993.118} C_VEL
LIN {X 0,Y 540.452,Z 867.565,A -85,B 0,C 180,E1 22992.268,E2 22992.268} C_VEL
LIN {X 0,Y 552.375,Z 873.838,A -85,B 0,C 180,E1 22991.463,E2 22991.463} C_VEL
LIN {X 0,Y 559.102,Z 876.388,A -85,B 0,C 180,E1 22991.003,E2 22991.003} C_VEL
LIN {X 0,Y 564.003,Z 877.346,A -85,B 0,C 180,E1 22990.49,E2 22990.49} C_VEL
LIN {X 0,Y 567.209,Z 877.364,A -85,B 0,C 180,E1 22989.969,E2 22989.969} C_VEL
LIN {X 0,Y 561.939,Z 890.73,A -85,B 0,C 180,E1 22989.644,E2 22989.644} C_VEL
LIN {X 0,Y 551.629,Z 909.461,A -85,B 0,C 180,E1 22989.453,E2 22989.453} C_VEL
LIN {X 0,Y 539.951,Z 928.246,A -85,B 0,C 180,E1 22989.082,E2 22989.082} C_VEL
LIN {X 0,Y 527.494,Z 948.386,A -85,B 0,C 180,E1 22988.479,E2 22988.479} C_VEL
LIN {X 0,Y 519.657,Z 963.763,A -85,B 0,C 180,E1 22987.934,E2 22987.934} C_VEL
LIN {X 0,Y 515.16,Z 975.044,A -85,B 0,C 180,E1 22987.479,E2 22987.479} C_VEL
LIN {X 0,Y 508.204,Z 989.383,A -85,B 0,C 180,E1 22986.946,E2 22986.946} C_VEL
LIN {X 0,Y 499.485,Z 1014.953,A -85,B 0,C 180,E1 22985.84,E2 22985.84} C_VEL
LIN {X 0,Y 497.757,Z 1021.787,A -85,B 0,C 180,E1 22985.554,E2 22985.554} C_VEL
LIN {X 0,Y 497.295,Z 1039.112,A -85,B 0,C 180,E1 22985.314,E2 22985.314} C_VEL
LIN {X 0,Y 496.77,Z 1068.472,A -85,B 0,C 180,E1 22984.822,E2 22984.822} C_VEL
LIN {X 0,Y 495.86,Z 1092.197,A -85,B 0,C 180,E1 22984.213,E2 22984.213} C_VEL
LIN {X 0,Y 494.789,Z 1115.693,A -85,B 0,C 180,E1 22983.378,E2 22983.378} C_VEL
LIN {X 0,Y 493.447,Z 1138.643,A -85,B 0,C 180,E1 22982.333,E2 22982.333} C_VEL
LIN {X 0,Y 492.193,Z 1157.526,A -85,B 0,C 180,E1 22981.268,E2 22981.268} C_VEL
LIN {X 0,Y 490.779,Z 1174.344,A -85,B 0,C 180,E1 22980.078,E2 22980.078} C_VEL
LIN {X 0,Y 488.86,Z 1193.545,A -85,B 0,C 180,E1 22978.422,E2 22978.422} C_VEL
LIN {X 0,Y 487.173,Z 1209.699,A -85,B 0,C 180,E1 22976.776,E2 22976.776} C_VEL
LIN {X 0,Y 485.7,Z 1224.163,A -85,B 0,C 180,E1 22975.092,E2 22975.092} C_VEL
LIN {X 0,Y 484.078,Z 1240.718,A -85,B 0,C 180,E1 22972.85,E2 22972.85} C_VEL
LIN {X 0,Y 482.915,Z 1253.254,A -85,B 0,C 180,E1 22970.863,E2 22970.863} C_VEL
LIN {X 0,Y 482.007,Z 1264.168,A -85,B 0,C 180,E1 22968.881,E2 22968.881} C_VEL
LIN {X 0,Y 481.132,Z 1276.315,A -85,B 0,C 180,E1 22966.293,E2 22966.293} C_VEL
LIN {X 0,Y 480.596,Z 1285.347,A -85,B 0,C 180,E1 22963.966,E2 22963.966} C_VEL
LIN {X 0,Y 480.244,Z 1293.208,A -85,B 0,C 180,E1 22961.53,E2 22961.53} C_VEL
LIN {X 0,Y 480.031,Z 1299.883,A -85,B 0,C 180,E1 22958.867,E2 22958.867} C_VEL
LIN {X 0,Y 479.95,Z 1304.188,A -85,B 0,C 180,E1 22956.58,E2 22956.58} C_VEL
LIN {X 0,Y 479.905,Z 1307.491,A -85,B 0,C 180,E1 22954.063,E2 22954.063} C_VEL
LIN {X 0,Y 479.9,Z 1309.201,A -85,B 0,C 180,E1 22951.433,E2 22951.433} C_VEL
LIN {X 0,Y 479.901,Z 1309.336,A -85,B 0,C 180,E1 22949.165,E2 22949.165} C_VEL
LIN {X 0,Y 479.908,Z 1308.272,A -85,B 0,C 180,E1 22946.895,E2 22946.895} C_VEL
LIN {X 0,Y 479.933,Z 1305.506,A -85,B 0,C 180,E1 22944.261,E2 22944.261} C_VEL
LIN {X 0,Y 479.995,Z 1300.995,A -85,B 0,C 180,E1 22941.669,E2 22941.669} C_VEL
LIN {X 0,Y 480.135,Z 1296.133,A -85,B 0,C 180,E1 22939.562,E2 22939.562} C_VEL
LIN {X 0,Y 480.412,Z 1289.129,A -85,B 0,C 180,E1 22937.133,E2 22937.133} C_VEL
LIN {X 0,Y 480.899,Z 1279.84,A -85,B 0,C 180,E1 22934.567,E2 22934.567} C_VEL
LIN {X 0,Y 481.546,Z 1270.21,A -85,B 0,C 180,E1 22932.354,E2 22932.354} C_VEL
LIN {X 0,Y 482.508,Z 1258.318,A -85,B 0,C 180,E1 22930.007,E2 22930.007} C_VEL
LIN {X 0,Y 483.686,Z 1244.827,A -85,B 0,C 180,E1 22927.773,E2 22927.773} C_VEL
LIN {X 0,Y 484.922,Z 1231.842,A -85,B 0,C 180,E1 22925.905,E2 22925.905} C_VEL
LIN {X 0,Y 486.571,Z 1215.966,A -85,B 0,C 180,E1 22923.913,E2 22923.913} C_VEL
LIN {X 0,Y 488.435,Z 1197.727,A -85,B 0,C 180,E1 22921.979,E2 22921.979} C_VEL
LIN {X 0,Y 490.321,Z 1179.055,A -85,B 0,C 180,E1 22920.297,E2 22920.297} C_VEL
LIN {X 0,Y 491.831,Z 1162.393,A -85,B 0,C 180,E1 22919.048,E2 22919.048} C_VEL
LIN {X 0,Y 493.409,Z 1142.081,A -85,B 0,C 180,E1 22917.796,E2 22917.796} C_VEL
LIN {X 0,Y 494.899,Z 1120.446,A -85,B 0,C 180,E1 22916.704,E2 22916.704} C_VEL
LIN {X 0,Y 496.242,Z 1098.049,A -85,B 0,C 180,E1 22915.812,E2 22915.812} C_VEL
LIN {X 0,Y 497.386,Z 1074.46,A -85,B 0,C 180,E1 22915.11,E2 22915.11} C_VEL
LIN {X 0,Y 498.157,Z 1050.793,A -85,B 0,C 180,E1 22914.637,E2 22914.637} C_VEL
LIN {X 0,Y 498.709,Z 1023.062,A -85,B 0,C 180,E1 22914.203,E2 22914.203} C_VEL
LIN {X 0,Y 503.323,Z 1007.891,A -85,B 0,C 180,E1 22913.491,E2 22913.491} C_VEL
LIN {X 0,Y 510.02,Z 989.155,A -85,B 0,C 180,E1 22912.716,E2 22912.716} C_VEL
LIN {X 0,Y 517.158,Z 973.704,A -85,B 0,C 180,E1 22912.203,E2 22912.203} C_VEL
LIN {X 0,Y 522.71,Z 959.992,A -85,B 0,C 180,E1 22911.702,E2 22911.702} C_VEL
LIN {X 0,Y 531.58,Z 942.809,A -85,B 0,C 180,E1 22911.22,E2 22911.22} C_VEL
LIN {X 0,Y 549.115,Z 913.668,A -85,B 0,C 180,E1 22910.613,E2 22910.613} C_VEL
LIN {X 0,Y 559.805,Z 894.862,A -85,B 0,C 180,E1 22910.385,E2 22910.385} C_VEL
LIN {X 0,Y 562.446,Z 889.527,A -85,B 0,C 180,E1 22910.33,E2 22910.33} C_VEL
LIN {X 0,Y 567.275,Z 877.187,A -85,B 0,C 180,E1 22910.026,E2 22910.026} C_VEL
LIN {X 0,Y 563.361,Z 877.292,A -85,B 0,C 180,E1 22909.43,E2 22909.43} C_VEL
LIN {X 0,Y 558.355,Z 876.185,A -85,B 0,C 180,E1 22908.928,E2 22908.928} C_VEL
LIN {X 0,Y 547.454,Z 872.172,A -85,B 0,C 180,E1 22907.86,E2 22907.86} C_VEL
LIN {X 0,Y 537.439,Z 866.526,A -85,B 0,C 180,E1 22906.67,E2 22906.67} C_VEL
LIN {X 0,Y 528.343,Z 858.992,A -85,B 0,C 180,E1 22905.361,E2 22905.361} C_VEL
LIN {X 0,Y 520.86,Z 849.915,A -85,B 0,C 180,E1 22904.019,E2 22904.019} C_VEL
LIN {X 0,Y 515.41,Z 840.182,A -85,B 0,C 180,E1 22902.763,E2 22902.763} C_VEL
LIN {X 0,Y 511.241,Z 828.721,A -85,B 0,C 180,E1 22901.454,E2 22901.454} C_VEL
LIN {X 0,Y 508.532,Z 815.432,A -85,B 0,C 180,E1 22900.108,E2 22900.108} C_VEL
LIN {X 0,Y 507.356,Z 799.731,A -85,B 0,C 180,E1 22898.703,E2 22898.703} C_VEL
LIN {X 0,Y 508.064,Z 780.157,A -85,B 0,C 180,E1 22897.154,E2 22897.154} C_VEL
LIN {X 0,Y 511.501,Z 739.614,A -85,B 0,C 180,E1 22894.081,E2 22894.081} C_VEL
LIN {X 0,Y 512.112,Z 731.873,A -85,B 0,C 180,E1 22893.474,E2 22893.474} C_VEL
LIN {X 0,Y 502.157,Z 713.311,A -85,B 0,C 180,E1 22890.381,E2 22890.381} C_VEL
LIN {X 0,Y 494.085,Z 698.815,A -85,B 0,C 180,E1 22887.738,E2 22887.738} C_VEL
LIN {X 0,Y 488.56,Z 689.07,A -85,B 0,C 180,E1 22885.843,E2 22885.843} C_VEL
LIN {X 0,Y 486.032,Z 684.531,A -85,B 0,C 180,E1 22884.943,E2 22884.943} C_VEL
LIN {X 0,Y 484.121,Z 681.354,A -85,B 0,C 180,E1 22884.267,E2 22884.267} C_VEL
LIN {X 0,Y 483.257,Z 679.595,A -85,B 0,C 180,E1 22883.924,E2 22883.924} C_VEL
LIN {X 0,Y 481.302,Z 676.552,A -85,B 0,C 180,E1 22883.247,E2 22883.247} C_VEL
LIN {X 0,Y 480.889,Z 674.833,A -85,B 0,C 180,E1 22882.963,E2 22882.963} C_VEL
LIN {X 0,Y 480.882,Z 674.834,A -85,B 0,C 180,E1 22879.431,E2 22879.431} C_VEL
LIN {X 0,Y 480.888,Z 674.833,A -85,B 0,C 180,E1 22875.805,E2 22875.805} C_VEL
LIN {X 0,Y 480.889,Z 674.833,A -85,B 0,C 180,E1 22872.122,E2 22872.122} C_VEL
LIN {X 0,Y 480.881,Z 674.833,A -85,B 0,C 180,E1 22868.61,E2 22868.61} C_VEL
LIN {X 0,Y 480.887,Z 674.833,A -85,B 0,C 180,E1 22865.01,E2 22865.01} C_VEL
LIN {X 0,Y 480.888,Z 674.836,A -85,B 0,C 180,E1 22861.31,E2 22861.31} C_VEL
LIN {X 0,Y 480.88,Z 674.836,A -85,B 0,C 180,E1 22857.736,E2 22857.736} C_VEL
LIN {X 0,Y 480.894,Z 674.832,A -85,B 0,C 180,E1 22854.033,E2 22854.033} C_VEL
LIN {X 0,Y 480.892,Z 674.836,A -85,B 0,C 180,E1 22850.304,E2 22850.304} C_VEL
LIN {X 0,Y 480.886,Z 674.831,A -85,B 0,C 180,E1 22846.656,E2 22846.656} C_VEL
LIN {X 0,Y 480.893,Z 674.834,A -85,B 0,C 180,E1 22842.952,E2 22842.952} C_VEL
LIN {X 0,Y 480.895,Z 674.835,A -85,B 0,C 180,E1 22839.301,E2 22839.301} C_VEL
LIN {X 0,Y 480.885,Z 674.832,A -85,B 0,C 180,E1 22835.558,E2 22835.558} C_VEL
LIN {X 0,Y 480.891,Z 674.801,A -85,B 0,C 180,E1 22831.972,E2 22831.972} C_VEL
LIN {X 0,Y 480.893,Z 674.834,A -85,B 0,C 180,E1 22828.252,E2 22828.252} C_VEL
LIN {X 0,Y 480.876,Z 674.803,A -85,B 0,C 180,E1 22824.592,E2 22824.592} C_VEL
LIN {X 0,Y 480.892,Z 674.83,A -85,B 0,C 180,E1 22821.041,E2 22821.041} C_VEL
LIN {X 0,Y 480.889,Z 674.833,A -85,B 0,C 180,E1 22817.327,E2 22817.327} C_VEL
LIN {X 0,Y 480.882,Z 674.841,A -85,B 0,C 180,E1 22813.818,E2 22813.818} C_VEL
LIN {X 0,Y 480.914,Z 675.018,A -85,B 0,C 180,E1 22813.401,E2 22813.401} C_VEL
LIN {X 0,Y 482.367,Z 678.572,A -85,B 0,C 180,E1 22812.97,E2 22812.97} C_VEL
LIN {X 0,Y 489.95,Z 695.135,A -85,B 0,C 180,E1 22810.888,E2 22810.888} C_VEL
LIN {X 0,Y 497.487,Z 713.263,A -85,B 0,C 180,E1 22808.737,E2 22808.737} C_VEL
LIN {X 0,Y 495.702,Z 751.264,A -85,B 0,C 180,E1 22805.967,E2 22805.967} C_VEL
LIN {X 0,Y 494.632,Z 756.243,A -85,B 0,C 180,E1 22805.694,E2 22805.694} C_VEL
LIN {X 0,Y 489.599,Z 767.88,A -85,B 0,C 180,E1 22805.327,E2 22805.327} C_VEL
LIN {X 0,Y 488.931,Z 772.593,A -85,B 0,C 180,E1 22805.19,E2 22805.19} C_VEL
LIN {X 0,Y 489.009,Z 773.268,A -85,B 0,C 180,E1 22805.169,E2 22805.169} C_VEL
LIN {X 0,Y 491.158,Z 788.44,A -85,B 0,C 180,E1 22804.723,E2 22804.723} C_VEL
LIN {X 0,Y 487.237,Z 1022.71,A -85,B 0,C 180,E1 22800.985,E2 22800.985} C_VEL
LIN {X 0,Y 486.627,Z 1043.354,A -85,B 0,C 180,E1 22800.531,E2 22800.531} C_VEL
LIN {X 0,Y 485.686,Z 1063.365,A -85,B 0,C 180,E1 22799.88,E2 22799.88} C_VEL
LIN {X 0,Y 484.484,Z 1083.142,A -85,B 0,C 180,E1 22799.011,E2 22799.011} C_VEL
LIN {X 0,Y 483.108,Z 1101.747,A -85,B 0,C 180,E1 22797.969,E2 22797.969} C_VEL
LIN {X 0,Y 481.572,Z 1119.968,A -85,B 0,C 180,E1 22796.711,E2 22796.711} C_VEL
LIN {X 0,Y 479.915,Z 1137.773,A -85,B 0,C 180,E1 22795.217,E2 22795.217} C_VEL
LIN {X 0,Y 478.271,Z 1154.403,A -85,B 0,C 180,E1 22793.534,E2 22793.534} C_VEL
LIN {X 0,Y 476.749,Z 1169.521,A -85,B 0,C 180,E1 22791.708,E2 22791.708} C_VEL
LIN {X 0,Y 475.418,Z 1182.941,A -85,B 0,C 180,E1 22789.791,E2 22789.791} C_VEL
LIN {X 0,Y 474.252,Z 1195.609,A -85,B 0,C 180,E1 22787.646,E2 22787.646} C_VEL
LIN {X 0,Y 473.311,Z 1207.071,A -85,B 0,C 180,E1 22785.31,E2 22785.31} C_VEL
LIN {X 0,Y 472.663,Z 1216.538,A -85,B 0,C 180,E1 22782.957,E2 22782.957} C_VEL
LIN {X 0,Y 472.257,Z 1224.156,A -85,B 0,C 180,E1 22780.614,E2 22780.614} C_VEL
